# B&R Automation Studio project TD52 (part 49)

```iecst
	xMsg36[73].Enable	:=	IN_CU.tPB2MM.bParaSetupOk ;
	xMsg36[73].Set		:=	OUT_CU.bMsg3673;(* B3673 reserve operating message *)
	IF xMsg36[73].Set THEN iReset_Msg36[73] := iDelay_MsgAutoReset_100ms; ELSE iReset_Msg36[73] := LIMIT(0, iReset_Msg36[73] -1,32767); END_IF		(* activate 'Message Hold Time' to avoid log clathering by repeated OpMsg entries *)
	xMsg36[73].Reset 	:= 	(iReset_Msg36[73] < 1);		//.Reset := TRUE;
	xMsg36[73]();
	MM2VIS.bMsg3673		:=	xMsg36[73].Q;

	xMsg36[74].Enable	:=	IN_CU.tPB2MM.bParaSetupOk ;
	xMsg36[74].Set		:=	OUT_CU.bMsg3674;(* B3674 reserve operating message *)
	IF xMsg36[74].Set THEN iReset_Msg36[74] := iDelay_MsgAutoReset_100ms; ELSE iReset_Msg36[74] := LIMIT(0, iReset_Msg36[74] -1,32767); END_IF		(* activate 'Message Hold Time' to avoid log clathering by repeated OpMsg entries *)
	xMsg36[74].Reset 	:= 	(iReset_Msg36[74] < 1);		//.Reset := TRUE;
	xMsg36[74]();
	MM2VIS.bMsg3674		:=	xMsg36[74].Q;

	xMsg36[75].Enable	:=	IN_CU.tPB2MM.bParaSetupOk ;
	xMsg36[75].Set		:=	OUT_CU.bMsg3675;(* B3675 reserve operating message *)
	IF xMsg36[75].Set THEN iReset_Msg36[75] := iDelay_MsgAutoReset_100ms; ELSE iReset_Msg36[75] := LIMIT(0, iReset_Msg36[75] -1,32767); END_IF		(* activate 'Message Hold Time' to avoid log clathering by repeated OpMsg entries *)
	xMsg36[75].Reset 	:= 	(iReset_Msg36[75] < 1);		//.Reset := TRUE;
	xMsg36[75]();
	MM2VIS.bMsg3675		:=	xMsg36[75].Q;

	xMsg36[76].Enable	:=	IN_CU.tPB2MM.bParaSetupOk ;
	xMsg36[76].Set		:=	OUT_CU.bMsg3676;(* B3676 reserve operating message *)
	IF xMsg36[76].Set THEN iReset_Msg36[76] := iDelay_MsgAutoReset_100ms; ELSE iReset_Msg36[76] := LIMIT(0, iReset_Msg36[76] -1,32767); END_IF		(* activate 'Message Hold Time' to avoid log clathering by repeated OpMsg entries *)
	xMsg36[76].Reset 	:= 	(iReset_Msg36[76] < 1);		//.Reset := TRUE;
	xMsg36[76]();
	MM2VIS.bMsg3676		:=	xMsg36[76].Q;

	xMsg36[77].Enable	:=	IN_CU.tPB2MM.bParaSetupOk ;
	xMsg36[77].Set		:=	OUT_CU.bMsg3677;(* B3677 reserve operating message *)
	IF xMsg36[77].Set THEN iReset_Msg36[77] := iDelay_MsgAutoReset_100ms; ELSE iReset_Msg36[77] := LIMIT(0, iReset_Msg36[77] -1,32767); END_IF		(* activate 'Message Hold Time' to avoid log clathering by repeated OpMsg entries *)
	xMsg36[77].Reset 	:= 	(iReset_Msg36[77] < 1);		//.Reset := TRUE;
	xMsg36[77]();
	MM2VIS.bMsg3677		:=	xMsg36[77].Q;

	xMsg36[78].Enable	:=	IN_CU.tPB2MM.bParaSetupOk ;
	xMsg36[78].Set		:=	OUT_CU.bMsg3678;(* B3678 reserve operating message *)
	IF xMsg36[78].Set THEN iReset_Msg36[78] := iDelay_MsgAutoReset_100ms; ELSE iReset_Msg36[78] := LIMIT(0, iReset_Msg36[78] -1,32767); END_IF		(* activate 'Message Hold Time' to avoid log clathering by repeated OpMsg entries *)
	xMsg36[78].Reset 	:= 	(iReset_Msg36[78] < 1);		//.Reset := TRUE;
	xMsg36[78]();
	MM2VIS.bMsg3678		:=	xMsg36[78].Q;

	xMsg36[79].Enable	:=	IN_CU.tPB2MM.bParaSetupOk ;
	xMsg36[79].Set		:=	OUT_CU.bMsg3679;(* B3679 reserve operating message *)
	IF xMsg36[79].Set THEN iReset_Msg36[79] := iDelay_MsgAutoReset_100ms; ELSE iReset_Msg36[79] := LIMIT(0, iReset_Msg36[79] -1,32767); END_IF		(* activate 'Message Hold Time' to avoid log clathering by repeated OpMsg entries *)
	xMsg36[79].Reset 	:= 	(iReset_Msg36[79] < 1);		//.Reset := TRUE;
	xMsg36[79]();
	MM2VIS.bMsg3679		:=	xMsg36[79].Q;

	xMsg36[80].Enable	:=	IN_CU.tPB2MM.bParaSetupOk ;
	xMsg36[80].Set		:=	OUT_CU.bMsg3680;(* B3680 reserve operating message *)
	IF xMsg36[80].Set THEN iReset_Msg36[80] := iDelay_MsgAutoReset_100ms; ELSE iReset_Msg36[80] := LIMIT(0, iReset_Msg36[80] -1,32767); END_IF		(* activate 'Message Hold Time' to avoid log clathering by repeated OpMsg entries *)
	xMsg36[80].Reset 	:= 	(iReset_Msg36[80] < 1);		//.Reset := TRUE;
	xMsg36[80]();
	MM2VIS.bMsg3680		:=	xMsg36[80].Q;
	(*----------------------------------------------------------------------*)

	xMsg36[81].Enable	:=	IN_CU.tPB2MM.bParaSetupOk ;
	xMsg36[81].Set		:=	OUT_CU.bMsg3681;(* B3681 reserve operating message *)
	IF xMsg36[81].Set THEN iReset_Msg36[81] := iDelay_MsgAutoReset_100ms; ELSE iReset_Msg36[81] := LIMIT(0, iReset_Msg36[81] -1,32767); END_IF		(* activate 'Message Hold Time' to avoid log clathering by repeated OpMsg entries *)
	xMsg36[81].Reset 	:= 	(iReset_Msg36[81] < 1);		//.Reset := TRUE;
	xMsg36[81]();
	MM2VIS.bMsg3681		:=	xMsg36[81].Q;

	xMsg36[82].Enable	:=	IN_CU.tPB2MM.bParaSetupOk ;
	xMsg36[82].Set		:=	OUT_CU.bMsg3682;(* B3682 reserve operating message *)
	IF xMsg36[82].Set THEN iReset_Msg36[82] := iDelay_MsgAutoReset_100ms; ELSE iReset_Msg36[82] := LIMIT(0, iReset_Msg36[82] -1,32767); END_IF		(* activate 'Message Hold Time' to avoid log clathering by repeated OpMsg entries *)
	xMsg36[82].Reset 	:= 	(iReset_Msg36[82] < 1);		//.Reset := TRUE;
	xMsg36[82]();
	MM2VIS.bMsg3682		:=	xMsg36[82].Q;

	xMsg36[83].Enable	:=	IN_CU.tPB2MM.bParaSetupOk ;
	xMsg36[83].Set		:=	OUT_CU.bMsg3683;(* B3683 reserve operating message *)
	IF xMsg36[83].Set THEN iReset_Msg36[83] := iDelay_MsgAutoReset_100ms; ELSE iReset_Msg36[83] := LIMIT(0, iReset_Msg36[83] -1,32767); END_IF		(* activate 'Message Hold Time' to avoid log clathering by repeated OpMsg entries *)
	xMsg36[83].Reset 	:= 	(iReset_Msg36[83] < 1);		//.Reset := TRUE;
	xMsg36[83]();
	MM2VIS.bMsg3683		:=	xMsg36[83].Q;

	xMsg36[84].Enable	:=	IN_CU.tPB2MM.bParaSetupOk ;
	xMsg36[84].Set		:=	OUT_CU.bMsg3684;(* B3684 reserve operating message *)
	IF xMsg36[84].Set THEN iReset_Msg36[84] := iDelay_MsgAutoReset_100ms; ELSE iReset_Msg36[84] := LIMIT(0, iReset_Msg36[84] -1,32767); END_IF		(* activate 'Message Hold Time' to avoid log clathering by repeated OpMsg entries *)
	xMsg36[84].Reset 	:= 	(iReset_Msg36[84] < 1);		//.Reset := TRUE;
	xMsg36[84]();
	MM2VIS.bMsg3684		:=	xMsg36[84].Q;

	xMsg36[85].Enable	:=	IN_CU.tPB2MM.bParaSetupOk ;
	xMsg36[85].Set		:=	OUT_CU.bMsg3685;(* B3685 reserve operating message *)
	IF xMsg36[85].Set THEN iReset_Msg36[85] := iDelay_MsgAutoReset_100ms; ELSE iReset_Msg36[85] := LIMIT(0, iReset_Msg36[85] -1,32767); END_IF		(* activate 'Message Hold Time' to avoid log clathering by repeated OpMsg entries *)
	xMsg36[85].Reset 	:= 	(iReset_Msg36[85] < 1);		//.Reset := TRUE;
	xMsg36[85]();
	MM2VIS.bMsg3685		:=	xMsg36[85].Q;

	xMsg36[86].Enable	:=	IN_CU.tPB2MM.bParaSetupOk ;
	xMsg36[86].Set		:=	OUT_CU.bMsg3686;(* B3686 reserve operating message *)
	IF xMsg36[86].Set THEN iReset_Msg36[86] := iDelay_MsgAutoReset_100ms; ELSE iReset_Msg36[86] := LIMIT(0, iReset_Msg36[86] -1,32767); END_IF		(* activate 'Message Hold Time' to avoid log clathering by repeated OpMsg entries *)
	xMsg36[86].Reset 	:= 	(iReset_Msg36[86] < 1);		//.Reset := TRUE;
	xMsg36[86]();
	MM2VIS.bMsg3686		:=	xMsg36[86].Q;

	xMsg36[87].Enable	:=	IN_CU.tPB2MM.bParaSetupOk ;
	xMsg36[87].Set		:=	OUT_CU.bMsg3687;(* B3687 reserve operating message *)
	IF xMsg36[87].Set THEN iReset_Msg36[87] := iDelay_MsgAutoReset_100ms; ELSE iReset_Msg36[87] := LIMIT(0, iReset_Msg36[87] -1,32767); END_IF		(* activate 'Message Hold Time' to avoid log clathering by repeated OpMsg entries *)
	xMsg36[87].Reset 	:= 	(iReset_Msg36[87] < 1);		//.Reset := TRUE;
	xMsg36[87]();
	MM2VIS.bMsg3687		:=	xMsg36[87].Q;

	xMsg36[88].Enable	:=	IN_CU.tPB2MM.bParaSetupOk ;
	xMsg36[88].Set		:=	OUT_CU.bMsg3688;(* B3688 reserve operating message *)
	IF xMsg36[88].Set THEN iReset_Msg36[88] := iDelay_MsgAutoReset_100ms; ELSE iReset_Msg36[88] := LIMIT(0, iReset_Msg36[88] -1,32767); END_IF		(* activate 'Message Hold Time' to avoid log clathering by repeated OpMsg entries *)
	xMsg36[88].Reset 	:= 	(iReset_Msg36[88] < 1);		//.Reset := TRUE;
	xMsg36[88]();
	MM2VIS.bMsg3688		:=	xMsg36[88].Q;

	xMsg36[89].Enable	:=	IN_CU.tPB2MM.bParaSetupOk ;
	xMsg36[89].Set		:=	OUT_CU.bMsg3689;(* B3689 reserve operating message *)
	IF xMsg36[89].Set THEN iReset_Msg36[89] := iDelay_MsgAutoReset_100ms; ELSE iReset_Msg36[89] := LIMIT(0, iReset_Msg36[89] -1,32767); END_IF		(* activate 'Message Hold Time' to avoid log clathering by repeated OpMsg entries *)
	xMsg36[89].Reset 	:= 	(iReset_Msg36[89] < 1);		//.Reset := TRUE;
	xMsg36[89]();
	MM2VIS.bMsg3689		:=	xMsg36[89].Q;

	xMsg36[90].Enable	:=	IN_CU.tPB2MM.bParaSetupOk ;
	xMsg36[90].Set		:=	OUT_CU.bMsg3690;(* B3690 reserve operating message *)
	IF xMsg36[90].Set THEN iReset_Msg36[90] := iDelay_MsgAutoReset_100ms; ELSE iReset_Msg36[90] := LIMIT(0, iReset_Msg36[90] -1,32767); END_IF		(* activate 'Message Hold Time' to avoid log clathering by repeated OpMsg entries *)
	xMsg36[90].Reset 	:= 	(iReset_Msg36[90] < 1);		//.Reset := TRUE;
	xMsg36[90]();
	MM2VIS.bMsg3690		:=	xMsg36[90].Q;
	(*----------------------------------------------------------------------*)

	xMsg36[91].Enable	:=	IN_CU.tPB2MM.bParaSetupOk ;
	xMsg36[91].Set		:=	OUT_CU.bMsg3691;(* B3691 reserve operating message *)
	IF xMsg36[91].Set THEN iReset_Msg36[91] := iDelay_MsgAutoReset_100ms; ELSE iReset_Msg36[91] := LIMIT(0, iReset_Msg36[91] -1,32767); END_IF		(* activate 'Message Hold Time' to avoid log clathering by repeated OpMsg entries *)
	xMsg36[91].Reset 	:= 	(iReset_Msg36[91] < 1);		//.Reset := TRUE;
	xMsg36[91]();
	MM2VIS.bMsg3691		:=	xMsg36[91].Q;

	xMsg36[92].Enable	:=	IN_CU.tPB2MM.bParaSetupOk ;
	xMsg36[92].Set		:=	OUT_CU.bMsg3692;(* B3692 reserve operating message *)
	IF xMsg36[92].Set THEN iReset_Msg36[92] := iDelay_MsgAutoReset_100ms; ELSE iReset_Msg36[92] := LIMIT(0, iReset_Msg36[92] -1,32767); END_IF		(* activate 'Message Hold Time' to avoid log clathering by repeated OpMsg entries *)
	xMsg36[92].Reset 	:= 	(iReset_Msg36[92] < 1);		//.Reset := TRUE;
	xMsg36[92]();
	MM2VIS.bMsg3692		:=	xMsg36[92].Q;

	xMsg36[93].Enable	:=	IN_CU.tPB2MM.bParaSetupOk ;
	xMsg36[93].Set		:=	OUT_CU.bMsg3693;(* B3693 reserve operating message *)
	IF xMsg36[93].Set THEN iReset_Msg36[93] := iDelay_MsgAutoReset_100ms; ELSE iReset_Msg36[93] := LIMIT(0, iReset_Msg36[93] -1,32767); END_IF		(* activate 'Message Hold Time' to avoid log clathering by repeated OpMsg entries *)
	xMsg36[93].Reset 	:= 	(iReset_Msg36[93] < 1);		//.Reset := TRUE;
	xMsg36[93]();
	MM2VIS.bMsg3693		:=	xMsg36[93].Q;

	xMsg36[94].Enable	:=	IN_CU.tPB2MM.bParaSetupOk ;
	xMsg36[94].Set		:=	OUT_CU.bMsg3694;(* B3694 reserve operating message *)
	IF xMsg36[94].Set THEN iReset_Msg36[94] := iDelay_MsgAutoReset_100ms; ELSE iReset_Msg36[94] := LIMIT(0, iReset_Msg36[94] -1,32767); END_IF		(* activate 'Message Hold Time' to avoid log clathering by repeated OpMsg entries *)
	xMsg36[94].Reset 	:= 	(iReset_Msg36[94] < 1);		//.Reset := TRUE;
	xMsg36[94]();
	MM2VIS.bMsg3694		:=	xMsg36[94].Q;

	xMsg36[95].Enable	:=	IN_CU.tPB2MM.bParaSetupOk ;
	xMsg36[95].Set		:=	OUT_CU.bMsg3695;(* B3695 reserve operating message *)
	IF xMsg36[95].Set THEN iReset_Msg36[95] := iDelay_MsgAutoReset_100ms; ELSE iReset_Msg36[95] := LIMIT(0, iReset_Msg36[95] -1,32767); END_IF		(* activate 'Message Hold Time' to avoid log clathering by repeated OpMsg entries *)
	xMsg36[95].Reset 	:= 	(iReset_Msg36[95] < 1);		//.Reset := TRUE;
	xMsg36[95]();
	MM2VIS.bMsg3695		:=	xMsg36[95].Q;

	xMsg36[96].Enable	:=	IN_CU.tPB2MM.bParaSetupOk ;
	xMsg36[96].Set		:=	OUT_CU.bMsg3696;(* B3696 reserve operating message *)
	IF xMsg36[96].Set THEN iReset_Msg36[96] := iDelay_MsgAutoReset_100ms; ELSE iReset_Msg36[96] := LIMIT(0, iReset_Msg36[96] -1,32767); END_IF		(* activate 'Message Hold Time' to avoid log clathering by repeated OpMsg entries *)
	xMsg36[96].Reset 	:= 	(iReset_Msg36[96] < 1);		//.Reset := TRUE;
	xMsg36[96]();
	MM2VIS.bMsg3696		:=	xMsg36[96].Q;

	xMsg36[97].Enable	:=	IN_CU.tPB2MM.bParaSetupOk ;
	xMsg36[97].Set		:=	OUT_CU.bMsg3697;(* B3697 reserve operating message *)
	IF xMsg36[97].Set THEN iReset_Msg36[97] := iDelay_MsgAutoReset_100ms; ELSE iReset_Msg36[97] := LIMIT(0, iReset_Msg36[97] -1,32767); END_IF		(* activate 'Message Hold Time' to avoid log clathering by repeated OpMsg entries *)
	xMsg36[97].Reset 	:= 	(iReset_Msg36[97] < 1);		//.Reset := TRUE;
	xMsg36[97]();
	MM2VIS.bMsg3697		:=	xMsg36[97].Q;

	xMsg36[98].Enable	:=	IN_CU.tPB2MM.bParaSetupOk ;
	xMsg36[98].Set		:=	OUT_CU.bMsg3698;(* B3698 reserve operating message *)
	IF xMsg36[98].Set THEN iReset_Msg36[98] := iDelay_MsgAutoReset_100ms; ELSE iReset_Msg36[98] := LIMIT(0, iReset_Msg36[98] -1,32767); END_IF		(* activate 'Message Hold Time' to avoid log clathering by repeated OpMsg entries *)
	xMsg36[98].Reset 	:= 	(iReset_Msg36[98] < 1);		//.Reset := TRUE;
	xMsg36[98]();
	MM2VIS.bMsg3698		:=	xMsg36[98].Q;

	xMsg36[99].Enable	:=	IN_CU.tPB2MM.bParaSetupOk ;
	xMsg36[99].Set		:=	OUT_CU.bMsg3699;(* B3699 reserve operating message *)
	IF xMsg36[99].Set THEN iReset_Msg36[99] := iDelay_MsgAutoReset_100ms; ELSE iReset_Msg36[99] := LIMIT(0, iReset_Msg36[99] -1,32767); END_IF		(* activate 'Message Hold Time' to avoid log clathering by repeated OpMsg entries *)
	xMsg36[99].Reset 	:= 	(iReset_Msg36[99] < 1);		//.Reset := TRUE;
	xMsg36[99]();
	MM2VIS.bMsg3699		:=	xMsg36[99].Q;

	xMsg3700.Enable		:=	IN_CU.tPB2MM.bParaSetupOk ;
	xMsg3700.Set		:=	OUT_CU.bMsg3700;(* B3700 reserve operating message *)
	IF xMsg3700.Set THEN iReset_Msg3700 := iDelay_MsgAutoReset_100ms; ELSE iReset_Msg3700 := LIMIT(0, iReset_Msg3700 -1,32767); END_IF		(* activate 'Message Hold Time' to avoid log clathering by repeated OpMsg entries *)
	xMsg3700.Reset 	:= 	(iReset_Msg3700 < 1);		//.Reset := TRUE;
	xMsg3700();
	MM2VIS.bMsg3700		:=	xMsg3700.Q;

	(* W6701 to W6799:  reserve operating message 109 - 207 *) (*import HMI Extension *)
	FOR cnt := 01 TO 99 DO
		(*set standard message options*)
		xMsg67[cnt].Enable	:= 	IN_CU.tPB2MM.bParaSetupOk ;
		IF xMsg67[cnt].Set THEN iReset_Msg67[cnt] := iDelay_MsgAutoReset_100ms; ELSE iReset_Msg67[cnt] := LIMIT(0, iReset_Msg67[cnt] -1,32767); END_IF		(* activate 'Message Hold Time' to avoid log clathering by repeated OpMsg entries *)
		xMsg67[cnt].Reset 	:= 	(iReset_Msg67[cnt] < 1);		//.Reset := TRUE;
		xMsg67[cnt]();	(*function call*)
	END_FOR

	xMsg67[01].Set		:=	OUT_CU.bMsg6701;(* B6701 reserve operating message 109 *) (*import HMI Extension *)
	MM2VIS.bMsg6701		:=	xMsg67[01].Q;

	xMsg67[02].Set		:=	OUT_CU.bMsg6702;(* B6702 reserve operating message 110 *) (*import HMI Extension *)
	MM2VIS.bMsg6702		:=	xMsg67[02].Q;

	xMsg67[03].Set		:=	OUT_CU.bMsg6703;(* B6703 reserve operating message 111 *) (*import HMI Extension *)
	MM2VIS.bMsg6703		:=	xMsg67[03].Q;

	xMsg67[04].Set		:=	OUT_CU.bMsg6704;(* B6704 reserve operating message 112 *) (*import HMI Extension *)
	MM2VIS.bMsg6704		:=	xMsg67[04].Q;

	xMsg67[05].Set		:=	OUT_CU.bMsg6705;(* B6705 reserve operating message 113 *) (*import HMI Extension *)
	MM2VIS.bMsg6705		:=	xMsg67[05].Q;

	xMsg67[06].Set		:=	OUT_CU.bMsg6706;(* B6706 reserve operating message 114 *) (*import HMI Extension *)
	MM2VIS.bMsg6706		:=	xMsg67[06].Q;

	xMsg67[07].Set		:=	OUT_CU.bMsg6707;(* B6707 reserve operating message 115 *) (*import HMI Extension *)
	MM2VIS.bMsg6707		:=	xMsg67[07].Q;

	xMsg67[08].Set		:=	OUT_CU.bMsg6708;(* B6708 reserve operating message 116 *) (*import HMI Extension *)
	MM2VIS.bMsg6708		:=	xMsg67[08].Q;

	xMsg67[09].Set		:=	OUT_CU.bMsg6709;(* B6709 reserve operating message 117 *) (*import HMI Extension *)
	MM2VIS.bMsg6709		:=	xMsg67[09].Q;

	xMsg67[10].Set		:=	OUT_CU.bMsg6710;(* B6710 reserve operating message 118 *) (*import HMI Extension *)
	MM2VIS.bMsg6710		:=	xMsg67[10].Q;

	xMsg67[11].Set		:=	OUT_CU.bMsg6711;(* B6711 reserve operating message 119 *) (*import HMI Extension *)
	MM2VIS.bMsg6711		:=	xMsg67[11].Q;

	xMsg67[12].Set		:=	OUT_CU.bMsg6712;(* B6712 reserve operating message 120 *) (*import HMI Extension *)
	MM2VIS.bMsg6712		:=	xMsg67[12].Q;

	xMsg67[13].Set		:=	OUT_CU.bMsg6713;(* B6713 reserve operating message 121 *) (*import HMI Extension *)
	MM2VIS.bMsg6713		:=	xMsg67[13].Q;

	xMsg67[14].Set		:=	OUT_CU.bMsg6714;(* B6714 reserve operating message 122 *) (*import HMI Extension *)
	MM2VIS.bMsg6714		:=	xMsg67[14].Q;

	xMsg67[15].Set		:=	OUT_CU.bMsg6715;(* B6715 reserve operating message 123 *) (*import HMI Extension *)
	MM2VIS.bMsg6715		:=	xMsg67[15].Q;

	xMsg67[16].Set		:=	OUT_CU.bMsg6716;(* B6716 reserve operating message 124 *) (*import HMI Extension *)
	MM2VIS.bMsg6716		:=	xMsg67[16].Q;

	xMsg67[17].Set		:=	OUT_CU.bMsg6717;(* B6717 reserve operating message 125 *) (*import HMI Extension *)
	MM2VIS.bMsg6717		:=	xMsg67[17].Q;

	xMsg67[18].Set		:=	OUT_CU.bMsg6718;(* B6718 reserve operating message 126 *) (*import HMI Extension *)
	MM2VIS.bMsg6718		:=	xMsg67[18].Q;

	xMsg67[19].Set		:=	OUT_CU.bMsg6719;(* B6719 reserve operating message 127 *) (*import HMI Extension *)
	MM2VIS.bMsg6719		:=	xMsg67[19].Q;

	xMsg67[20].Set		:=	OUT_CU.bMsg6720;(* B6720 reserve operating message 128 *) (*import HMI Extension *)
	MM2VIS.bMsg6720		:=	xMsg67[20].Q;

	xMsg67[21].Set		:=	OUT_CU.bMsg6721;(* B6721 reserve operating message 129 *) (*import HMI Extension *)
	MM2VIS.bMsg6721		:=	xMsg67[21].Q;

	xMsg67[22].Set		:=	OUT_CU.bMsg6722;(* B6722 reserve operating message 130 *) (*import HMI Extension *)
	MM2VIS.bMsg6722		:=	xMsg67[22].Q;

	xMsg67[23].Set		:=	OUT_CU.bMsg6723;(* B6723 reserve operating message 131 *) (*import HMI Extension *)
	MM2VIS.bMsg6723		:=	xMsg67[23].Q;

	xMsg67[24].Set		:=	OUT_CU.bMsg6724;(* B6724 reserve operating message 132 *) (*import HMI Extension *)
	MM2VIS.bMsg6724		:=	xMsg67[24].Q;

	xMsg67[25].Set		:=	OUT_CU.bMsg6725;(* B6725 reserve operating message 133 *) (*import HMI Extension *)
	MM2VIS.bMsg6725		:=	xMsg67[25].Q;

	xMsg67[26].Set		:=	OUT_CU.bMsg6726;(* B6726 reserve operating message 134 *) (*import HMI Extension *)
	MM2VIS.bMsg6726		:=	xMsg67[26].Q;

	xMsg67[27].Set		:=	OUT_CU.bMsg6727;(* B6727 reserve operating message 135 *) (*import HMI Extension *)
	MM2VIS.bMsg6727		:=	xMsg67[27].Q;

	xMsg67[28].Set		:=	OUT_CU.bMsg6728;(* B6728 reserve operating message 136 *) (*import HMI Extension *)
	MM2VIS.bMsg6728		:=	xMsg67[28].Q;

	xMsg67[29].Set		:=	OUT_CU.bMsg6729;(* B6729 reserve operating message 137 *) (*import HMI Extension *)
	MM2VIS.bMsg6729		:=	xMsg67[29].Q;

	xMsg67[30].Set		:=	OUT_CU.bMsg6730;(* B6730 reserve operating message 138 *) (*import HMI Extension *)
	MM2VIS.bMsg6730		:=	xMsg67[30].Q;

	xMsg67[31].Set		:=	OUT_CU.bMsg6731;(* B6731 reserve operating message 139 *) (*import HMI Extension *)
	MM2VIS.bMsg6731		:=	xMsg67[31].Q;

	xMsg67[32].Set		:=	OUT_CU.bMsg6732;(* B6732 reserve operating message 140 *) (*import HMI Extension *)
	MM2VIS.bMsg6732		:=	xMsg67[32].Q;

	xMsg67[33].Set		:=	OUT_CU.bMsg6733;(* B6733 reserve operating message 141 *) (*import HMI Extension *)
	MM2VIS.bMsg6733		:=	xMsg67[33].Q;

	xMsg67[34].Set		:=	OUT_CU.bMsg6734;(* B6734 reserve operating message 142 *) (*import HMI Extension *)
	MM2VIS.bMsg6734		:=	xMsg67[34].Q;

	xMsg67[35].Set		:=	OUT_CU.bMsg6735;(* B6735 reserve operating message 143 *) (*import HMI Extension *)
	MM2VIS.bMsg6735		:=	xMsg67[35].Q;

	xMsg67[36].Set		:=	OUT_CU.bMsg6736;(* B6736 reserve operating message 144 *) (*import HMI Extension *)
	MM2VIS.bMsg6736		:=	xMsg67[36].Q;

	xMsg67[37].Set		:=	OUT_CU.bMsg6737;(* B6737 reserve operating message 145 *) (*import HMI Extension *)
	MM2VIS.bMsg6737		:=	xMsg67[37].Q;

	xMsg67[38].Set		:=	OUT_CU.bMsg6738;(* B6738 reserve operating message 146 *) (*import HMI Extension *)
	MM2VIS.bMsg6738		:=	xMsg67[38].Q;

	xMsg67[39].Set		:=	OUT_CU.bMsg6739;(* B6739 reserve operating message 147 *) (*import HMI Extension *)
	MM2VIS.bMsg6739		:=	xMsg67[39].Q;

	xMsg67[40].Set		:=	OUT_CU.bMsg6740;(* B6740 reserve operating message 148 *) (*import HMI Extension *)
	MM2VIS.bMsg6740		:=	xMsg67[40].Q;

	xMsg67[41].Set		:=	OUT_CU.bMsg6741;(* B6741 reserve operating message 149 *) (*import HMI Extension *)
	MM2VIS.bMsg6741		:=	xMsg67[41].Q;

	xMsg67[42].Set		:=	OUT_CU.bMsg6742;(* B6742 reserve operating message 150 *) (*import HMI Extension *)
	MM2VIS.bMsg6742		:=	xMsg67[42].Q;

	xMsg67[43].Set		:=	OUT_CU.bMsg6743;(* B6743 reserve operating message 151 *) (*import HMI Extension *)
	MM2VIS.bMsg6743		:=	xMsg67[43].Q;

	xMsg67[44].Set		:=	OUT_CU.bMsg6744;(* B6744 reserve operating message 152 *) (*import HMI Extension *)
	MM2VIS.bMsg6744		:=	xMsg67[44].Q;

	xMsg67[45].Set		:=	OUT_CU.bMsg6745;(* B6745 reserve operating message 153 *) (*import HMI Extension *)
	MM2VIS.bMsg6745		:=	xMsg67[45].Q;

	xMsg67[46].Set		:=	OUT_CU.bMsg6746;(* B6746 reserve operating message 154 *) (*import HMI Extension *)
	MM2VIS.bMsg6746		:=	xMsg67[46].Q;

	xMsg67[47].Set		:=	OUT_CU.bMsg6747;(* B6747 reserve operating message 155 *) (*import HMI Extension *)
	MM2VIS.bMsg6747		:=	xMsg67[47].Q;

	xMsg67[48].Set		:=	OUT_CU.bMsg6748;(* B6748 reserve operating message 156 *) (*import HMI Extension *)
	MM2VIS.bMsg6748		:=	xMsg67[48].Q;

	xMsg67[49].Set		:=	OUT_CU.bMsg6749;(* B6749 reserve operating message 157 *) (*import HMI Extension *)
	MM2VIS.bMsg6749		:=	xMsg67[49].Q;

	xMsg67[50].Set		:=	OUT_CU.bMsg6750;(* B6750 reserve operating message 158 *) (*import HMI Extension *)
	MM2VIS.bMsg6750		:=	xMsg67[50].Q;

	xMsg67[51].Set		:=	OUT_CU.bMsg6751;(* B6751 reserve operating message 159 *) (*import HMI Extension *)
	MM2VIS.bMsg6751		:=	xMsg67[51].Q;

	xMsg67[52].Set		:=	OUT_CU.bMsg6752;(* B6752 reserve operating message 160 *) (*import HMI Extension *)
	MM2VIS.bMsg6752		:=	xMsg67[52].Q;

	xMsg67[53].Set		:=	OUT_CU.bMsg6753;(* B6753 reserve operating message 161 *) (*import HMI Extension *)
	MM2VIS.bMsg6753		:=	xMsg67[53].Q;

	xMsg67[54].Set		:=	OUT_CU.bMsg6754;(* B6754 reserve operating message 162 *) (*import HMI Extension *)
	MM2VIS.bMsg6754		:=	xMsg67[54].Q;

	xMsg67[55].Set		:=	OUT_CU.bMsg6755;(* B6755 reserve operating message 163 *) (*import HMI Extension *)
	MM2VIS.bMsg6755		:=	xMsg67[55].Q;

	xMsg67[56].Set		:=	OUT_CU.bMsg6756;(* B6756 reserve operating message 164 *) (*import HMI Extension *)
	MM2VIS.bMsg6756		:=	xMsg67[56].Q;

	xMsg67[57].Set		:=	OUT_CU.bMsg6757;(* B6757 reserve operating message 165 *) (*import HMI Extension *)
	MM2VIS.bMsg6757		:=	xMsg67[57].Q;

	xMsg67[58].Set		:=	OUT_CU.bMsg6758;(* B6758 reserve operating message 166 *) (*import HMI Extension *)
	MM2VIS.bMsg6758		:=	xMsg67[58].Q;

	xMsg67[59].Set		:=	OUT_CU.bMsg6759;(* B6759 reserve operating message 167 *) (*import HMI Extension *)
	MM2VIS.bMsg6759		:=	xMsg67[59].Q;

	xMsg67[60].Set		:=	OUT_CU.bMsg6760;(* B6760 reserve operating message 168 *) (*import HMI Extension *)
	MM2VIS.bMsg6760		:=	xMsg67[60].Q;

	xMsg67[61].Set		:=	OUT_CU.bMsg6761;(* B6761 reserve operating message 169 *) (*import HMI Extension *)
	MM2VIS.bMsg6761		:=	xMsg67[61].Q;

	xMsg67[62].Set		:=	OUT_CU.bMsg6762;(* B6762 reserve operating message 170 *) (*import HMI Extension *)
	MM2VIS.bMsg6762		:=	xMsg67[62].Q;

	xMsg67[63].Set		:=	OUT_CU.bMsg6763;(* B6763 reserve operating message 171 *) (*import HMI Extension *)
	MM2VIS.bMsg6763		:=	xMsg67[63].Q;

	xMsg67[64].Set		:=	OUT_CU.bMsg6764;(* B6764 reserve operating message 172 *) (*import HMI Extension *)
	MM2VIS.bMsg6764		:=	xMsg67[64].Q;

	xMsg67[65].Set		:=	OUT_CU.bMsg6765;(* B6765 reserve operating message 173 *) (*import HMI Extension *)
	MM2VIS.bMsg6765		:=	xMsg67[65].Q;

	xMsg67[66].Set		:=	OUT_CU.bMsg6766;(* B6766 reserve operating message 174 *) (*import HMI Extension *)
	MM2VIS.bMsg6766		:=	xMsg67[66].Q;

	xMsg67[67].Set		:=	OUT_CU.bMsg6767;(* B6767 reserve operating message 175 *) (*import HMI Extension *)
	MM2VIS.bMsg6767		:=	xMsg67[67].Q;

	xMsg67[68].Set		:=	OUT_CU.bMsg6768;(* B6768 reserve operating message 176 *) (*import HMI Extension *)
	MM2VIS.bMsg6768		:=	xMsg67[68].Q;

	xMsg67[69].Set		:=	OUT_CU.bMsg6769;(* B6769 reserve operating message 177 *) (*import HMI Extension *)
	MM2VIS.bMsg6769		:=	xMsg67[69].Q;

	xMsg67[70].Set		:=	OUT_CU.bMsg6770;(* B6770 reserve operating message 178 *) (*import HMI Extension *)
	MM2VIS.bMsg6770		:=	xMsg67[70].Q;

	xMsg67[71].Set		:=	OUT_CU.bMsg6771;(* B6771 reserve operating message 179 *) (*import HMI Extension *)
	MM2VIS.bMsg6771		:=	xMsg67[71].Q;

	xMsg67[72].Set		:=	OUT_CU.bMsg6772;(* B6772 reserve operating message 180 *) (*import HMI Extension *)
	MM2VIS.bMsg6772		:=	xMsg67[72].Q;

	xMsg67[73].Set		:=	OUT_CU.bMsg6773;(* B6773 reserve operating message 181 *) (*import HMI Extension *)
	MM2VIS.bMsg6773		:=	xMsg67[73].Q;

	xMsg67[74].Set		:=	OUT_CU.bMsg6774;(* B6774 reserve operating message 182 *) (*import HMI Extension *)
	MM2VIS.bMsg6774		:=	xMsg67[74].Q;

	xMsg67[75].Set		:=	OUT_CU.bMsg6775;(* B6775 reserve operating message 183 *) (*import HMI Extension *)
	MM2VIS.bMsg6775		:=	xMsg67[75].Q;

	xMsg67[76].Set		:=	OUT_CU.bMsg6776;(* B6776 reserve operating message 184 *) (*import HMI Extension *)
	MM2VIS.bMsg6776		:=	xMsg67[76].Q;

	xMsg67[77].Set		:=	OUT_CU.bMsg6777;(* B6777 reserve operating message 185 *) (*import HMI Extension *)
	MM2VIS.bMsg6777		:=	xMsg67[77].Q;

	xMsg67[78].Set		:=	OUT_CU.bMsg6778;(* B6778 reserve operating message 186 *) (*import HMI Extension *)
	MM2VIS.bMsg6778		:=	xMsg67[78].Q;

	xMsg67[79].Set		:=	OUT_CU.bMsg6779;(* B6779 reserve operating message 187 *) (*import HMI Extension *)
	MM2VIS.bMsg6779		:=	xMsg67[79].Q;

	xMsg67[80].Set		:=	OUT_CU.bMsg6780;(* B6780 reserve operating message 188 *) (*import HMI Extension *)
	MM2VIS.bMsg6780		:=	xMsg67[80].Q;

	xMsg67[81].Set		:=	OUT_CU.bMsg6781;(* B6781 reserve operating message 189 *) (*import HMI Extension *)
	MM2VIS.bMsg6781		:=	xMsg67[81].Q;

	xMsg67[82].Set		:=	OUT_CU.bMsg6782;(* B6782 reserve operating message 190 *) (*import HMI Extension *)
	MM2VIS.bMsg6782		:=	xMsg67[82].Q;

	xMsg67[83].Set		:=	OUT_CU.bMsg6783;(* B6783 reserve operating message 191 *) (*import HMI Extension *)
	MM2VIS.bMsg6783		:=	xMsg67[83].Q;

	xMsg67[84].Set		:=	OUT_CU.bMsg6784;(* B6784 reserve operating message 192 *) (*import HMI Extension *)
	MM2VIS.bMsg6784		:=	xMsg67[84].Q;

	xMsg67[85].Set		:=	OUT_CU.bMsg6785;(* B6785 reserve operating message 193 *) (*import HMI Extension *)
	MM2VIS.bMsg6785		:=	xMsg67[85].Q;

	xMsg67[86].Set		:=	OUT_CU.bMsg6786;(* B6786 reserve operating message 194 *) (*import HMI Extension *)
	MM2VIS.bMsg6786		:=	xMsg67[86].Q;

	xMsg67[87].Set		:=	OUT_CU.bMsg6787;(* B6787 reserve operating message 195 *) (*import HMI Extension *)
	MM2VIS.bMsg6787		:=	xMsg67[87].Q;

	xMsg67[88].Set		:=	OUT_CU.bMsg6788;(* B6788 reserve operating message 196 *) (*import HMI Extension *)
	MM2VIS.bMsg6788		:=	xMsg67[88].Q;

	xMsg67[89].Set		:=	OUT_CU.bMsg6789;(* B6789 reserve operating message 197 *) (*import HMI Extension *)
	MM2VIS.bMsg6789		:=	xMsg67[89].Q;

	xMsg67[90].Set		:=	OUT_CU.bMsg6790;(* B6790 reserve operating message 198 *) (*import HMI Extension *)
	MM2VIS.bMsg6790		:=	xMsg67[90].Q;

	xMsg67[91].Set		:=	OUT_CU.bMsg6791;(* B6791 reserve operating message 199 *) (*import HMI Extension *)
	MM2VIS.bMsg6791		:=	xMsg67[91].Q;

	xMsg67[92].Set		:=	OUT_CU.bMsg6792;(* B6792 reserve operating message 200 *) (*import HMI Extension *)
	MM2VIS.bMsg6792		:=	xMsg67[92].Q;

	xMsg67[93].Set		:=	OUT_CU.bMsg6793;(* B6793 reserve operating message 201 *) (*import HMI Extension *)
	MM2VIS.bMsg6793		:=	xMsg67[93].Q;

	xMsg67[94].Set		:=	OUT_CU.bMsg6794;(* B6794 reserve operating message 202 *) (*import HMI Extension *)
	MM2VIS.bMsg6794		:=	xMsg67[94].Q;

	xMsg67[95].Set		:=	OUT_CU.bMsg6795;(* B6795 reserve operating message 203 *) (*import HMI Extension *)
	MM2VIS.bMsg6795		:=	xMsg67[95].Q;

	xMsg67[96].Set		:=	OUT_CU.bMsg6796;(* B6796 reserve operating message 204 *) (*import HMI Extension *)
	MM2VIS.bMsg6796		:=	xMsg67[96].Q;

	xMsg67[97].Set		:=	OUT_CU.bMsg6797;(* B6797 reserve operating message 205 *) (*import HMI Extension *)
	MM2VIS.bMsg6797		:=	xMsg67[97].Q;

	xMsg67[98].Set		:=	OUT_CU.bMsg6798;(* B6798 reserve operating message 206 *) (*import HMI Extension *)
	MM2VIS.bMsg6798		:=	xMsg67[98].Q;

	xMsg67[99].Set		:=	OUT_CU.bMsg6799;(* B6799 reserve operating message 207 *) (*import HMI Extension *)
	MM2VIS.bMsg6799		:=	xMsg67[99].Q;

//	xMsg67[100].Set		//	MOVED TO xMsg68[0].Set
//	MM2VIS.bMsg6800		//	MOVED TO xMsg68[0].Set

	(* W6800 to W6899:  reserve operating message 208 - 307 *) (*import HMI Extension *)
	FOR cnt := 00 TO 99 DO
		(*set standard message options*)
		xMsg68[cnt].Enable	:= 	IN_CU.tPB2MM.bParaSetupOk ;
		IF xMsg68[cnt].Set THEN iReset_Msg68[cnt] := iDelay_MsgAutoReset_100ms; ELSE iReset_Msg68[cnt] := LIMIT(0, iReset_Msg68[cnt] -1,32767); END_IF		(* activate 'Message Hold Time' to avoid log clathering by repeated OpMsg entries *)
		xMsg68[cnt].Reset 	:= 	(iReset_Msg68[cnt] < 1);		//.Reset := TRUE;
		xMsg68[cnt]();	(*function call*)
	END_FOR

	xMsg68[0].Set		:=	OUT_CU.bMsg6800;(* B6800 reserve operating message 208 *) (*import HMI Extension *)
	MM2VIS.bMsg6800		:=	xMsg68[0].Q;

	xMsg68[01].Set		:=	OUT_CU.bMsg6801;(* B6801 reserve operating message 209 *) (*import HMI Extension *)
	MM2VIS.bMsg6801		:=	xMsg68[01].Q;

	xMsg68[02].Set		:=	OUT_CU.bMsg6802;(* B6802 reserve operating message 210 *) (*import HMI Extension *)
	MM2VIS.bMsg6802		:=	xMsg68[02].Q;

	xMsg68[03].Set		:=	OUT_CU.bMsg6803;(* B6803 reserve operating message 211 *) (*import HMI Extension *)
	MM2VIS.bMsg6803		:=	xMsg68[03].Q;

	xMsg68[04].Set		:=	OUT_CU.bMsg6804;(* B6804 reserve operating message 212 *) (*import HMI Extension *)
	MM2VIS.bMsg6804		:=	xMsg68[04].Q;

	xMsg68[05].Set		:=	OUT_CU.bMsg6805;(* B6805 reserve operating message 213 *) (*import HMI Extension *)
	MM2VIS.bMsg6805		:=	xMsg68[05].Q;

	xMsg68[06].Set		:=	OUT_CU.bMsg6806;(* B6806 reserve operating message 214 *) (*import HMI Extension *)
	MM2VIS.bMsg6806		:=	xMsg68[06].Q;

	xMsg68[07].Set		:=	OUT_CU.bMsg6807;(* B6807 reserve operating message 215 *) (*import HMI Extension *)
	MM2VIS.bMsg6807		:=	xMsg68[07].Q;

	xMsg68[08].Set		:=	OUT_CU.bMsg6808;(* B6808 reserve operating message 216 *) (*import HMI Extension *)
	MM2VIS.bMsg6808		:=	xMsg68[08].Q;

	xMsg68[09].Set		:=	OUT_CU.bMsg6809;(* B6809 reserve operating message 217 *) (*import HMI Extension *)
	MM2VIS.bMsg6809		:=	xMsg68[09].Q;

	xMsg68[10].Set		:=	OUT_CU.bMsg6810;(* B6810 reserve operating message 218 *) (*import HMI Extension *)
	MM2VIS.bMsg6810		:=	xMsg68[10].Q;

	xMsg68[11].Set		:=	OUT_CU.bMsg6811;(* B6811 reserve operating message 219 *) (*import HMI Extension *)
	MM2VIS.bMsg6811		:=	xMsg68[11].Q;

	xMsg68[12].Set		:=	OUT_CU.bMsg6812;(* B6812 reserve operating message 220 *) (*import HMI Extension *)
	MM2VIS.bMsg6812		:=	xMsg68[12].Q;

	xMsg68[13].Set		:=	OUT_CU.bMsg6813;(* B6813 reserve operating message 221 *) (*import HMI Extension *)
	MM2VIS.bMsg6813		:=	xMsg68[13].Q;

	xMsg68[14].Set		:=	OUT_CU.bMsg6814;(* B6814 reserve operating message 222 *) (*import HMI Extension *)
	MM2VIS.bMsg6814		:=	xMsg68[14].Q;

	xMsg68[15].Set		:=	OUT_CU.bMsg6815;(* B6815 reserve operating message 223 *) (*import HMI Extension *)
	MM2VIS.bMsg6815		:=	xMsg68[15].Q;

	xMsg68[16].Set		:=	OUT_CU.bMsg6816;(* B6816 reserve operating message 224 *) (*import HMI Extension *)
	MM2VIS.bMsg6816		:=	xMsg68[16].Q;

	xMsg68[17].Set		:=	OUT_CU.bMsg6817;(* B6817 reserve operating message 225 *) (*import HMI Extension *)
	MM2VIS.bMsg6817		:=	xMsg68[17].Q;

	xMsg68[18].Set		:=	OUT_CU.bMsg6818;(* B6818 reserve operating message 226 *) (*import HMI Extension *)
	MM2VIS.bMsg6818		:=	xMsg68[18].Q;

	xMsg68[19].Set		:=	OUT_CU.bMsg6819;(* B6819 reserve operating message 227 *) (*import HMI Extension *)
	MM2VIS.bMsg6819		:=	xMsg68[19].Q;

	xMsg68[20].Set		:=	OUT_CU.bMsg6820;(* B6820 reserve operating message 228 *) (*import HMI Extension *)
	MM2VIS.bMsg6820		:=	xMsg68[20].Q;

	xMsg68[21].Set		:=	OUT_CU.bMsg6821;(* B6821 reserve operating message 229 *) (*import HMI Extension *)
	MM2VIS.bMsg6821		:=	xMsg68[21].Q;

	xMsg68[22].Set		:=	OUT_CU.bMsg6822;(* B6822 reserve operating message 230 *) (*import HMI Extension *)
	MM2VIS.bMsg6822		:=	xMsg68[22].Q;

	xMsg68[23].Set		:=	OUT_CU.bMsg6823;(* B6823 reserve operating message 231 *) (*import HMI Extension *)
	MM2VIS.bMsg6823		:=	xMsg68[23].Q;

	xMsg68[24].Set		:=	OUT_CU.bMsg6824;(* B6824 reserve operating message 232 *) (*import HMI Extension *)
	MM2VIS.bMsg6824		:=	xMsg68[24].Q;

	xMsg68[25].Set		:=	OUT_CU.bMsg6825;(* B6825 reserve operating message 233 *) (*import HMI Extension *)
	MM2VIS.bMsg6825		:=	xMsg68[25].Q;

	xMsg68[26].Set		:=	OUT_CU.bMsg6826;(* B6826 reserve operating message 234 *) (*import HMI Extension *)
	MM2VIS.bMsg6826		:=	xMsg68[26].Q;

	xMsg68[27].Set		:=	OUT_CU.bMsg6827;(* B6827 reserve operating message 235 *) (*import HMI Extension *)
	MM2VIS.bMsg6827		:=	xMsg68[27].Q;

	xMsg68[28].Set		:=	OUT_CU.bMsg6828;(* B6828 reserve operating message 236 *) (*import HMI Extension *)
	MM2VIS.bMsg6828		:=	xMsg68[28].Q;

	xMsg68[29].Set		:=	OUT_CU.bMsg6829;(* B6829 reserve operating message 237 *) (*import HMI Extension *)
	MM2VIS.bMsg6829		:=	xMsg68[29].Q;

	xMsg68[30].Set		:=	OUT_CU.bMsg6830;(* B6830 reserve operating message 238 *) (*import HMI Extension *)
	MM2VIS.bMsg6830		:=	xMsg68[30].Q;

	xMsg68[31].Set		:=	OUT_CU.bMsg6831;(* B6831 reserve operating message 239 *) (*import HMI Extension *)
	MM2VIS.bMsg6831		:=	xMsg68[31].Q;

	xMsg68[32].Set		:=	OUT_CU.bMsg6832;(* B6832 reserve operating message 240 *) (*import HMI Extension *)
	MM2VIS.bMsg6832		:=	xMsg68[32].Q;

	xMsg68[33].Set		:=	OUT_CU.bMsg6833;(* B6833 reserve operating message 241 *) (*import HMI Extension *)
	MM2VIS.bMsg6833		:=	xMsg68[33].Q;

	xMsg68[34].Set		:=	OUT_CU.bMsg6834;(* B6834 reserve operating message 242 *) (*import HMI Extension *)
	MM2VIS.bMsg6834		:=	xMsg68[34].Q;

	xMsg68[35].Set		:=	OUT_CU.bMsg6835;(* B6835 reserve operating message 243 *) (*import HMI Extension *)
	MM2VIS.bMsg6835		:=	xMsg68[35].Q;

	xMsg68[36].Set		:=	OUT_CU.bMsg6836;(* B6836 reserve operating message 244 *) (*import HMI Extension *)
	MM2VIS.bMsg6836		:=	xMsg68[36].Q;

	xMsg68[37].Set		:=	OUT_CU.bMsg6837;(* B6837 reserve operating message 245 *) (*import HMI Extension *)
	MM2VIS.bMsg6837		:=	xMsg68[37].Q;

	xMsg68[38].Set		:=	OUT_CU.bMsg6838;(* B6838 reserve operating message 246 *) (*import HMI Extension *)
	MM2VIS.bMsg6838		:=	xMsg68[38].Q;

	xMsg68[39].Set		:=	OUT_CU.bMsg6839;(* B6839 reserve operating message 247 *) (*import HMI Extension *)
	MM2VIS.bMsg6839		:=	xMsg68[39].Q;

	xMsg68[40].Set		:=	OUT_CU.bMsg6840;(* B6840 reserve operating message 248 *) (*import HMI Extension *)
	MM2VIS.bMsg6840		:=	xMsg68[40].Q;

	xMsg68[41].Set		:=	OUT_CU.bMsg6841;(* B6841 reserve operating message 249 *) (*import HMI Extension *)
	MM2VIS.bMsg6841		:=	xMsg68[41].Q;

	xMsg68[42].Set		:=	OUT_CU.bMsg6842;(* B6842 reserve operating message 250 *) (*import HMI Extension *)
	MM2VIS.bMsg6842		:=	xMsg68[42].Q;

	xMsg68[43].Set		:=	OUT_CU.bMsg6843;(* B6843 reserve operating message 251 *) (*import HMI Extension *)
	MM2VIS.bMsg6843		:=	xMsg68[43].Q;

	xMsg68[44].Set		:=	OUT_CU.bMsg6844;(* B6844 reserve operating message 252 *) (*import HMI Extension *)
	MM2VIS.bMsg6844		:=	xMsg68[44].Q;

	xMsg68[45].Set		:=	OUT_CU.bMsg6845;(* B6845 reserve operating message 253 *) (*import HMI Extension *)
	MM2VIS.bMsg6845		:=	xMsg68[45].Q;

	xMsg68[46].Set		:=	OUT_CU.bMsg6846;(* B6846 reserve operating message 254 *) (*import HMI Extension *)
	MM2VIS.bMsg6846		:=	xMsg68[46].Q;

	xMsg68[47].Set		:=	OUT_CU.bMsg6847;(* B6847 reserve operating message 255 *) (*import HMI Extension *)
	MM2VIS.bMsg6847		:=	xMsg68[47].Q;

	xMsg68[48].Set		:=	OUT_CU.bMsg6848;(* B6848 reserve operating message 256 *) (*import HMI Extension *)
	MM2VIS.bMsg6848		:=	xMsg68[48].Q;

	xMsg68[49].Set		:=	OUT_CU.bMsg6849;(* B6849 reserve operating message 257 *) (*import HMI Extension *)
	MM2VIS.bMsg6849		:=	xMsg68[49].Q;

	xMsg68[50].Set		:=	OUT_CU.bMsg6850;(* B6850 reserve operating message 258 *) (*import HMI Extension *)
	MM2VIS.bMsg6850		:=	xMsg68[50].Q;

	xMsg68[51].Set		:=	OUT_CU.bMsg6851;(* B6851 reserve operating message 259 *) (*import HMI Extension *)
	MM2VIS.bMsg6851		:=	xMsg68[51].Q;

	xMsg68[52].Set		:=	OUT_CU.bMsg6852;(* B6852 reserve operating message 260 *) (*import HMI Extension *)
	MM2VIS.bMsg6852		:=	xMsg68[52].Q;

	xMsg68[53].Set		:=	OUT_CU.bMsg6853;(* B6853 reserve operating message 261 *) (*import HMI Extension *)
	MM2VIS.bMsg6853		:=	xMsg68[53].Q;

	xMsg68[54].Set		:=	OUT_CU.bMsg6854;(* B6854 reserve operating message 262 *) (*import HMI Extension *)
	MM2VIS.bMsg6854		:=	xMsg68[54].Q;

	xMsg68[55].Set		:=	OUT_CU.bMsg6855;(* B6855 reserve operating message 263 *) (*import HMI Extension *)
	MM2VIS.bMsg6855		:=	xMsg68[55].Q;

	xMsg68[56].Set		:=	OUT_CU.bMsg6856;(* B6856 reserve operating message 264 *) (*import HMI Extension *)
	MM2VIS.bMsg6856		:=	xMsg68[56].Q;

	xMsg68[57].Set		:=	OUT_CU.bMsg6857;(* B6857 reserve operating message 265 *) (*import HMI Extension *)
	MM2VIS.bMsg6857		:=	xMsg68[57].Q;

	xMsg68[58].Set		:=	OUT_CU.bMsg6858;(* B6858 reserve operating message 266 *) (*import HMI Extension *)
	MM2VIS.bMsg6858		:=	xMsg68[58].Q;

	xMsg68[59].Set		:=	OUT_CU.bMsg6859;(* B6859 reserve operating message 267 *) (*import HMI Extension *)
	MM2VIS.bMsg6859		:=	xMsg68[59].Q;

	xMsg68[60].Set		:=	OUT_CU.bMsg6860;(* B6860 reserve operating message 268 *) (*import HMI Extension *)
	MM2VIS.bMsg6860		:=	xMsg68[60].Q;

	xMsg68[61].Set		:=	OUT_CU.bMsg6861;(* B6861 reserve operating message 269 *) (*import HMI Extension *)
	MM2VIS.bMsg6861		:=	xMsg68[61].Q;

	xMsg68[62].Set		:=	OUT_CU.bMsg6862;(* B6862 reserve operating message 270 *) (*import HMI Extension *)
	MM2VIS.bMsg6862		:=	xMsg68[62].Q;

	xMsg68[63].Set		:=	OUT_CU.bMsg6863;(* B6863 reserve operating message 271 *) (*import HMI Extension *)
	MM2VIS.bMsg6863		:=	xMsg68[63].Q;

	xMsg68[64].Set		:=	OUT_CU.bMsg6864;(* B6864 reserve operating message 272 *) (*import HMI Extension *)
	MM2VIS.bMsg6864		:=	xMsg68[64].Q;

	xMsg68[65].Set		:=	OUT_CU.bMsg6865;(* B6865 reserve operating message 273 *) (*import HMI Extension *)
	MM2VIS.bMsg6865		:=	xMsg68[65].Q;

	xMsg68[66].Set		:=	OUT_CU.bMsg6866;(* B6866 reserve operating message 274 *) (*import HMI Extension *)
	MM2VIS.bMsg6866		:=	xMsg68[66].Q;

	xMsg68[67].Set		:=	OUT_CU.bMsg6867;(* B6867 reserve operating message 275 *) (*import HMI Extension *)
	MM2VIS.bMsg6867		:=	xMsg68[67].Q;

	xMsg68[68].Set		:=	OUT_CU.bMsg6868;(* B6868 reserve operating message 276 *) (*import HMI Extension *)
	MM2VIS.bMsg6868		:=	xMsg68[68].Q;

	xMsg68[69].Set		:=	OUT_CU.bMsg6869;(* B6869 reserve operating message 277 *) (*import HMI Extension *)
	MM2VIS.bMsg6869		:=	xMsg68[69].Q;

	xMsg68[70].Set		:=	OUT_CU.bMsg6870;(* B6870 reserve operating message 278 *) (*import HMI Extension *)
	MM2VIS.bMsg6870		:=	xMsg68[70].Q;

	xMsg68[71].Set		:=	OUT_CU.bMsg6871;(* B6871 reserve operating message 279 *) (*import HMI Extension *)
	MM2VIS.bMsg6871		:=	xMsg68[71].Q;

	xMsg68[72].Set		:=	OUT_CU.bMsg6872;(* B6872 reserve operating message 280 *) (*import HMI Extension *)
	MM2VIS.bMsg6872		:=	xMsg68[72].Q;

	xMsg68[73].Set		:=	OUT_CU.bMsg6873;(* B6873 reserve operating message 281 *) (*import HMI Extension *)
	MM2VIS.bMsg6873		:=	xMsg68[73].Q;

	xMsg68[74].Set		:=	OUT_CU.bMsg6874;(* B6874 reserve operating message 282 *) (*import HMI Extension *)
	MM2VIS.bMsg6874		:=	xMsg68[74].Q;

	xMsg68[75].Set		:=	OUT_CU.bMsg6875;(* B6875 reserve operating message 283 *) (*import HMI Extension *)
	MM2VIS.bMsg6875		:=	xMsg68[75].Q;

	xMsg68[76].Set		:=	OUT_CU.bMsg6876;(* B6876 reserve operating message 284 *) (*import HMI Extension *)
	MM2VIS.bMsg6876		:=	xMsg68[76].Q;

	xMsg68[77].Set		:=	OUT_CU.bMsg6877;(* B6877 reserve operating message 285 *) (*import HMI Extension *)
	MM2VIS.bMsg6877		:=	xMsg68[77].Q;

	xMsg68[78].Set		:=	OUT_CU.bMsg6878;(* B6878 reserve operating message 286 *) (*import HMI Extension *)
	MM2VIS.bMsg6878		:=	xMsg68[78].Q;

	xMsg68[79].Set		:=	OUT_CU.bMsg6879;(* B6879 reserve operating message 287 *) (*import HMI Extension *)
	MM2VIS.bMsg6879		:=	xMsg68[79].Q;

	xMsg68[80].Set		:=	OUT_CU.bMsg6880;(* B6880 reserve operating message 288 *) (*import HMI Extension *)
	MM2VIS.bMsg6880		:=	xMsg68[80].Q;

	xMsg68[81].Set		:=	OUT_CU.bMsg6881;(* B6881 reserve operating message 289 *) (*import HMI Extension *)
	MM2VIS.bMsg6881		:=	xMsg68[81].Q;

	xMsg68[82].Set		:=	OUT_CU.bMsg6882;(* B6882 reserve operating message 290 *) (*import HMI Extension *)
	MM2VIS.bMsg6882		:=	xMsg68[82].Q;

	xMsg68[83].Set		:=	OUT_CU.bMsg6883;(* B6883 reserve operating message 291 *) (*import HMI Extension *)
	MM2VIS.bMsg6883		:=	xMsg68[83].Q;

	xMsg68[84].Set		:=	OUT_CU.bMsg6884;(* B6884 reserve operating message 292 *) (*import HMI Extension *)
	MM2VIS.bMsg6884		:=	xMsg68[84].Q;

	xMsg68[85].Set		:=	OUT_CU.bMsg6885;(* B6885 reserve operating message 293 *) (*import HMI Extension *)
	MM2VIS.bMsg6885		:=	xMsg68[85].Q;

	xMsg68[86].Set		:=	OUT_CU.bMsg6886;(* B6886 reserve operating message 294 *) (*import HMI Extension *)
	MM2VIS.bMsg6886		:=	xMsg68[86].Q;

	xMsg68[87].Set		:=	OUT_CU.bMsg6887;(* B6887 reserve operating message 295 *) (*import HMI Extension *)
	MM2VIS.bMsg6887		:=	xMsg68[87].Q;

	xMsg68[88].Set		:=	OUT_CU.bMsg6888;(* B6888 reserve operating message 296 *) (*import HMI Extension *)
	MM2VIS.bMsg6888		:=	xMsg68[88].Q;

	xMsg68[89].Set		:=	OUT_CU.bMsg6889;(* B6889 reserve operating message 297 *) (*import HMI Extension *)
	MM2VIS.bMsg6889		:=	xMsg68[89].Q;

	xMsg68[90].Set		:=	OUT_CU.bMsg6890;(* B6890 reserve operating message 298 *) (*import HMI Extension *)
	MM2VIS.bMsg6890		:=	xMsg68[90].Q;

	xMsg68[91].Set		:=	OUT_CU.bMsg6891;(* B6891 reserve operating message 299 *) (*import HMI Extension *)
	MM2VIS.bMsg6891		:=	xMsg68[91].Q;

	xMsg68[92].Set		:=	OUT_CU.bMsg6892;(* B6892 reserve operating message 300 *) (*import HMI Extension *)
	MM2VIS.bMsg6892		:=	xMsg68[92].Q;

	xMsg68[93].Set		:=	OUT_CU.bMsg6893;(* B6893 reserve operating message 301 *) (*import HMI Extension *)
	MM2VIS.bMsg6893		:=	xMsg68[93].Q;

	xMsg68[94].Set		:=	OUT_CU.bMsg6894;(* B6894 reserve operating message 302 *) (*import HMI Extension *)
	MM2VIS.bMsg6894		:=	xMsg68[94].Q;

	xMsg68[95].Set		:=	OUT_CU.bMsg6895;(* B6895 reserve operating message 303 *) (*import HMI Extension *)
	MM2VIS.bMsg6895		:=	xMsg68[95].Q;

	xMsg68[96].Set		:=	OUT_CU.bMsg6896;(* B6896 reserve operating message 304 *) (*import HMI Extension *)
	MM2VIS.bMsg6896		:=	xMsg68[96].Q;

	xMsg68[97].Set		:=	OUT_CU.bMsg6897;(* B6897 reserve operating message 305 *) (*import HMI Extension *)
	MM2VIS.bMsg6897		:=	xMsg68[97].Q;

	xMsg68[98].Set		:=	OUT_CU.bMsg6898;(* B6898 reserve operating message 306 *) (*import HMI Extension *)
	MM2VIS.bMsg6898		:=	xMsg68[98].Q;

	xMsg68[99].Set		:=	OUT_CU.bMsg6899;(* B6899 reserve operating message 307 *) (*import HMI Extension *)
	MM2VIS.bMsg6899		:=	xMsg68[99].Q;

//OLD	xMsg68[100].Set		:=	OUT_CU.bMsgxxxx;(* B4200 reserve operating message 308 OLD, do not use*) (*import HMI Extension *)
//OLD	MM2VIS.bMsg4200		:=	xMsg41[100].Q;

	(*----------------------------------------------------------------------*)
	iDelay_MsgAutoReset_100ms 	:= LIMIT(0, TIME_TO_INT(Para.tiDelay_MsgAutoReset / 100), 32767);	(*To Do: missing prototype parameter *)
	IF Para.tiDelay_MsgAutoReset = 0 THEN Para.tiDelay_MsgAutoReset := T#01m; END_IF				(*To Do: missing prototype parameter *)
	(*----------------------------------------------------------------------*)

END_PROGRAM
```

#### MsgCUInit.st - Initialization code
```iecst
(*******************************************************************************
Msg_CU	 			 alarms generation MM_Customized

This code is confidential and proprietary to the INNIO Company.
It may not be used in any form, or reproduced in any manner,
without written permission of the INNIO Company.
Copyright, INNIO Company, 2019

Customized modifications: -
------------------------

History:
-------
V0.00.0	29.07.2011	lettenb.	new
V4.07.1	29.03.2019	Hohensinner	added Warnings: W9285, W9286, W9287
V4.11.1	20.01.2022	Zengerer	added Arrays: B67xx, B68xx, W87xx

Instructions for use:
--------------------
1) declare alarm with function block "Msg"

2) use template to create a new alarm, substitue 0000 by message number:

	xMsg0000.Num		:=	0000;					alarm number
	xMsg0000.AmmSysAdr	:=  iAdrAmmBase2MM;			do not change
	xMsg0000.AmmOutAdr	:=  iAdrMM2AmmBase;			do not change

3) 	set alarm number

Outstandings:
------------
(*******************************************************************************)
PROGRAM _INIT

	iAdrAmmBase2MM		:=  ADR(IN_CU.tAB2CU);
	iAdrMM2AmmBase		:=  ADR(OUT_CU.tCU2AB);

	(*---------------------------------------------------------------------------*)
	xMsg1001.Num		:=	1001;
	xMsg1001.AmmInAdr	:=  iAdrAmmBase2MM;
	xMsg1001.AmmOutAdr	:=  iAdrMM2AmmBase;

	xMsg1002.Num		:=	1002;
	xMsg1002.AmmInAdr	:=  iAdrAmmBase2MM;
	xMsg1002.AmmOutAdr	:=  iAdrMM2AmmBase;

	xMsg1003.Num		:=	1003;
	xMsg1003.AmmInAdr	:=  iAdrAmmBase2MM;
	xMsg1003.AmmOutAdr	:=  iAdrMM2AmmBase;

	xMsg1004.Num		:=	1004;
	xMsg1004.AmmInAdr	:=  iAdrAmmBase2MM;
	xMsg1004.AmmOutAdr	:=  iAdrMM2AmmBase;

	xMsg1005.Num		:=	1005;
	xMsg1005.AmmInAdr	:=  iAdrAmmBase2MM;
	xMsg1005.AmmOutAdr	:=  iAdrMM2AmmBase;

	xMsg1006.Num		:=	1006;
	xMsg1006.AmmInAdr	:=  iAdrAmmBase2MM;
	xMsg1006.AmmOutAdr	:=  iAdrMM2AmmBase;

	xMsg1007.Num		:=	1007;
	xMsg1007.AmmInAdr	:=  iAdrAmmBase2MM;
	xMsg1007.AmmOutAdr	:=  iAdrMM2AmmBase;

	xMsg1008.Num		:=	1008;
	xMsg1008.AmmInAdr	:=  iAdrAmmBase2MM;
	xMsg1008.AmmOutAdr	:=  iAdrMM2AmmBase;

	xMsg1009.Num		:=	1009;
	xMsg1009.AmmInAdr	:=  iAdrAmmBase2MM;
	xMsg1009.AmmOutAdr	:=  iAdrMM2AmmBase;

	xMsg1010.Num		:=	1010;
	xMsg1010.AmmInAdr	:=  iAdrAmmBase2MM;
	xMsg1010.AmmOutAdr	:=  iAdrMM2AmmBase;

	xMsg1011.Num		:=	1011;
	xMsg1011.AmmInAdr	:=  iAdrAmmBase2MM;
	xMsg1011.AmmOutAdr	:=  iAdrMM2AmmBase;

	xMsg1012.Num		:=	1012;
	xMsg1012.AmmInAdr	:=  iAdrAmmBase2MM;
	xMsg1012.AmmOutAdr	:=  iAdrMM2AmmBase;

	xMsg1013.Num		:=	1013;
	xMsg1013.AmmInAdr	:=  iAdrAmmBase2MM;
	xMsg1013.AmmOutAdr	:=  iAdrMM2AmmBase;

	xMsg1014.Num		:=	1014;
	xMsg1014.AmmInAdr	:=  iAdrAmmBase2MM;
	xMsg1014.AmmOutAdr	:=  iAdrMM2AmmBase;

	xMsg1015.Num		:=	1015;
	xMsg1015.AmmInAdr	:=  iAdrAmmBase2MM;
	xMsg1015.AmmOutAdr	:=  iAdrMM2AmmBase;

	xMsg1016.Num		:=	1016;
	xMsg1016.AmmInAdr	:=  iAdrAmmBase2MM;
	xMsg1016.AmmOutAdr	:=  iAdrMM2AmmBase;

	xMsg1177.Num		:=	1177;			(* W1177 Signal fail: reserve analog in 1 *)
	xMsg1177.AmmInAdr	:=  iAdrAmmBase2MM;
	xMsg1177.AmmOutAdr	:=  iAdrMM2AmmBase;

	xMsg1178.Num		:=	1178;			(* W1178 Signal fail: reserve analog in 2 *)
	xMsg1178.AmmInAdr	:=  iAdrAmmBase2MM;
	xMsg1178.AmmOutAdr	:=  iAdrMM2AmmBase;

	xMsg1179.Num		:=	1179;			(* W1179 Signal fail: reserve analog in 3 *)
	xMsg1179.AmmInAdr	:=  iAdrAmmBase2MM;
	xMsg1179.AmmOutAdr	:=  iAdrMM2AmmBase;

	xMsg1180.Num		:=	1180;			(* W1180 Signal fail: reserve analog in 4 *)
	xMsg1180.AmmInAdr	:=  iAdrAmmBase2MM;
	xMsg1180.AmmOutAdr	:=  iAdrMM2AmmBase;

	xMsg1181.Num		:=	1181;			(* W1181 Signal fail: reserve analog in 5 *)
	xMsg1181.AmmInAdr	:=  iAdrAmmBase2MM;
	xMsg1181.AmmOutAdr	:=  iAdrMM2AmmBase;

	xMsg1182.Num		:=	1182;			(* W1182 Signal fail: reserve analog in 6 *)
	xMsg1182.AmmInAdr	:=  iAdrAmmBase2MM;
	xMsg1182.AmmOutAdr	:=  iAdrMM2AmmBase;

	xMsg1183.Num		:=	1183;			(* W1183 Signal fail: reserve analog in 7 *)
	xMsg1183.AmmInAdr	:=  iAdrAmmBase2MM;
	xMsg1183.AmmOutAdr	:=  iAdrMM2AmmBase;

	xMsg1184.Num		:=	1184;			(* W1184 Signal fail: reserve analog in 8 *)
	xMsg1184.AmmInAdr	:=  iAdrAmmBase2MM;
	xMsg1184.AmmOutAdr	:=  iAdrMM2AmmBase;

	xMsg1193.Num		:=	1193;
	xMsg1193.AmmInAdr	:=  iAdrAmmBase2MM;
	xMsg1193.AmmOutAdr	:=  iAdrMM2AmmBase;

	xMsg1194.Num		:=	1194;
	xMsg1194.AmmInAdr	:=  iAdrAmmBase2MM;
	xMsg1194.AmmOutAdr	:=  iAdrMM2AmmBase;

	xMsg1195.Num		:=	1195;
	xMsg1195.AmmInAdr	:=  iAdrAmmBase2MM;
	xMsg1195.AmmOutAdr	:=  iAdrMM2AmmBase;

	xMsg1196.Num		:=	1196;
	xMsg1196.AmmInAdr	:=  iAdrAmmBase2MM;
	xMsg1196.AmmOutAdr	:=  iAdrMM2AmmBase;

	xMsg1197.Num		:=	1197;
	xMsg1197.AmmInAdr	:=  iAdrAmmBase2MM;
	xMsg1197.AmmOutAdr	:=  iAdrMM2AmmBase;

	xMsg1198.Num		:=	1198;
	xMsg1198.AmmInAdr	:=  iAdrAmmBase2MM;
	xMsg1198.AmmOutAdr	:=  iAdrMM2AmmBase;

	xMsg1199.Num		:=	1199;
	xMsg1199.AmmInAdr	:=  iAdrAmmBase2MM;
	xMsg1199.AmmOutAdr	:=  iAdrMM2AmmBase;

	xMsg1200.Num		:=	1200;
	xMsg1200.AmmInAdr	:=  iAdrAmmBase2MM;
	xMsg1200.AmmOutAdr	:=  iAdrMM2AmmBase;

	xMsg1201.Num		:=	1201;
	xMsg1201.AmmInAdr	:=  iAdrAmmBase2MM;
	xMsg1201.AmmOutAdr	:=  iAdrMM2AmmBase;

	xMsg1202.Num		:=	1202;
	xMsg1202.AmmInAdr	:=  iAdrAmmBase2MM;
	xMsg1202.AmmOutAdr	:=  iAdrMM2AmmBase;

	xMsg1203.Num		:=	1203;
	xMsg1203.AmmInAdr	:=  iAdrAmmBase2MM;
	xMsg1203.AmmOutAdr	:=  iAdrMM2AmmBase;

	xMsg1204.Num		:=	1204;
	xMsg1204.AmmInAdr	:=  iAdrAmmBase2MM;
	xMsg1204.AmmOutAdr	:=  iAdrMM2AmmBase;

	xMsg1205.Num		:=	1205;
	xMsg1205.AmmInAdr	:=  iAdrAmmBase2MM;
	xMsg1205.AmmOutAdr	:=  iAdrMM2AmmBase;

	xMsg1206.Num		:=	1206;
	xMsg1206.AmmInAdr	:=  iAdrAmmBase2MM;
	xMsg1206.AmmOutAdr	:=  iAdrMM2AmmBase;

	xMsg1207.Num		:=	1207;
	xMsg1207.AmmInAdr	:=  iAdrAmmBase2MM;
	xMsg1207.AmmOutAdr	:=  iAdrMM2AmmBase;

	xMsg1208.Num		:=	1208;
	xMsg1208.AmmInAdr	:=  iAdrAmmBase2MM;
	xMsg1208.AmmOutAdr	:=  iAdrMM2AmmBase;

	(*W1300, W1301 - W1399 Reserve AnalogIN 1-30*)
	(*moved*)
	(*W1400, W1401 - W1499 Reserve AnalogIN ...*)
	(*moved*)

	(*A1601, A1602 - A1700 additional Reserve ALARMS *)
	FOR cnt := 0 TO 100 DO								(*remark: index 0 element is not in use, but called here also, to avoid possible watch errors in some AS- versions *)
		xMsg16[cnt].Num			:=	1600+cnt;
		xMsg16[cnt].AmmInAdr	:=  iAdrAmmBase2MM;
		xMsg16[cnt].AmmOutAdr	:=  iAdrMM2AmmBase;
	END_FOR

	(*W1701, W1702 - W1800 additional Reserve WARNINGS *)
	FOR cnt := 0 TO 100 DO								(*remark: index 0 element is not in use, but called here also, to avoid possible watch errors in some AS- versions *)
		xMsg17[cnt].Num			:=	1700+cnt;
		xMsg17[cnt].AmmInAdr	:=  iAdrAmmBase2MM;
		xMsg17[cnt].AmmOutAdr	:=  iAdrMM2AmmBase;
	END_FOR

	xMsg2087.Num		:=	2087;
	xMsg2087.AmmInAdr	:=  iAdrAmmBase2MM;
	xMsg2087.AmmOutAdr	:=  iAdrMM2AmmBase;

	xMsg2088.Num		:=	2088;
	xMsg2088.AmmInAdr	:=  iAdrAmmBase2MM;
	xMsg2088.AmmOutAdr	:=  iAdrMM2AmmBase;

	xMsg2089.Num		:=	2089;
	xMsg2089.AmmInAdr	:=  iAdrAmmBase2MM;
	xMsg2089.AmmOutAdr	:=  iAdrMM2AmmBase;

	xMsg2090.Num		:=	2090;
	xMsg2090.AmmInAdr	:=  iAdrAmmBase2MM;
	xMsg2090.AmmOutAdr	:=  iAdrMM2AmmBase;

	xMsg2091.Num		:=	2091;
	xMsg2091.AmmInAdr	:=  iAdrAmmBase2MM;
	xMsg2091.AmmOutAdr	:=  iAdrMM2AmmBase;

	xMsg2092.Num		:=	2092;
	xMsg2092.AmmInAdr	:=  iAdrAmmBase2MM;
	xMsg2092.AmmOutAdr	:=  iAdrMM2AmmBase;

	xMsg2093.Num		:=	2093;
	xMsg2093.AmmInAdr	:=  iAdrAmmBase2MM;
	xMsg2093.AmmOutAdr	:=  iAdrMM2AmmBase;

	xMsg2094.Num		:=	2094;
	xMsg2094.AmmInAdr	:=  iAdrAmmBase2MM;
	xMsg2094.AmmOutAdr	:=  iAdrMM2AmmBase;

	xMsg2095.Num		:=	2095;
	xMsg2095.AmmInAdr	:=  iAdrAmmBase2MM;
	xMsg2095.AmmOutAdr	:=  iAdrMM2AmmBase;

	xMsg2096.Num		:=	2096;
	xMsg2096.AmmInAdr	:=  iAdrAmmBase2MM;
	xMsg2096.AmmOutAdr	:=  iAdrMM2AmmBase;

	(*- NETZBEZUGSREGLER --------------------------------------------------------------------*)

	xMsg2302.Num		:=	2302;
	xMsg2302.AmmInAdr	:=  iAdrAmmBase2MM;
	xMsg2302.AmmOutAdr	:=  iAdrMM2AmmBase;

	xMsg2303.Num		:=	2303;
	xMsg2303.AmmInAdr	:=  iAdrAmmBase2MM;
	xMsg2303.AmmOutAdr	:=  iAdrMM2AmmBase;

	xMsg2415.Num		:=	2415;
	xMsg2415.AmmInAdr	:=  iAdrAmmBase2MM;
	xMsg2415.AmmOutAdr	:=  iAdrMM2AmmBase;

	xMsg2416.Num		:=	2416;
	xMsg2416.AmmInAdr	:=  iAdrAmmBase2MM;
	xMsg2416.AmmOutAdr	:=  iAdrMM2AmmBase;

	xMsg2417.Num		:=	2417;
	xMsg2417.AmmInAdr	:=  iAdrAmmBase2MM;
	xMsg2417.AmmOutAdr	:=  iAdrMM2AmmBase;

	xMsg2418.Num		:=	2418;
	xMsg2418.AmmInAdr	:=  iAdrAmmBase2MM;
	xMsg2418.AmmOutAdr	:=  iAdrMM2AmmBase;

	xMsg2419.Num		:=	2419;
	xMsg2419.AmmInAdr	:=  iAdrAmmBase2MM;
	xMsg2419.AmmOutAdr	:=  iAdrMM2AmmBase;

	xMsg2420.Num		:=	2420;
	xMsg2420.AmmInAdr	:=  iAdrAmmBase2MM;
	xMsg2420.AmmOutAdr	:=  iAdrMM2AmmBase;

	(*************)

	xMsg3232.Num		:=	3232;
	xMsg3232.AmmInAdr	:=  iAdrAmmBase2MM;
	xMsg3232.AmmOutAdr	:=  iAdrMM2AmmBase;

	xMsg3233.Num		:=	3233;
	xMsg3233.AmmInAdr	:=  iAdrAmmBase2MM;
	xMsg3233.AmmOutAdr	:=  iAdrMM2AmmBase;

	xMsg3234.Num		:=	3234;
	xMsg3234.AmmInAdr	:=  iAdrAmmBase2MM;
	xMsg3234.AmmOutAdr	:=  iAdrMM2AmmBase;

	xMsg3235.Num		:=	3235;
	xMsg3235.AmmInAdr	:=  iAdrAmmBase2MM;
	xMsg3235.AmmOutAdr	:=  iAdrMM2AmmBase;

	xMsg3236.Num		:=	3236;
	xMsg3236.AmmInAdr	:=  iAdrAmmBase2MM;
	xMsg3236.AmmOutAdr	:=  iAdrMM2AmmBase;

	xMsg3237.Num		:=	3237;
	xMsg3237.AmmInAdr	:=  iAdrAmmBase2MM;
	xMsg3237.AmmOutAdr	:=  iAdrMM2AmmBase;

	xMsg3250.Num		:=	3250;
	xMsg3250.AmmInAdr	:=  iAdrAmmBase2MM;
	xMsg3250.AmmOutAdr	:=  iAdrMM2AmmBase;

	xMsg3251.Num		:=	3251;
	xMsg3251.AmmInAdr	:=  iAdrAmmBase2MM;
	xMsg3251.AmmOutAdr	:=  iAdrMM2AmmBase;

	(*************)

	xMsg3565.Num		:=	3565;
	xMsg3565.AmmInAdr	:=  iAdrAmmBase2MM;
	xMsg3565.AmmOutAdr	:=  iAdrMM2AmmBase;

	(*************)

	(*A8966 - A8999 Reserve AnalogIN Alarms *)
	(*moved*)

	(*************)

	(*B3601 - 3699 additional Reserve op.messages *)
	FOR cnt := 0 TO 100 DO								(*remark: index 0 element is not in use, but called here also, to avoid possible watch errors in some AS- versions *)
		xMsg36[cnt].Num			:=	3600+cnt;			(* bugfix 2018! *)
		xMsg36[cnt].AmmInAdr	:=  iAdrAmmBase2MM;
		xMsg36[cnt].AmmOutAdr	:=  iAdrMM2AmmBase;
	END_FOR

	xMsg3700.Num		:=	3700;
	xMsg3700.AmmInAdr	:=  iAdrAmmBase2MM;
	xMsg3700.AmmOutAdr	:=  iAdrMM2AmmBase;

	(*B6701 - 6800 additional Reserve op.messages *)	(*import HMI Extension *)
	FOR cnt := 0 TO 100 DO								(*remark: index 0 element is not in use, but called here also, to avoid possible watch errors in some AS- versions *)
		xMsg67[cnt].Num			:=	6700+cnt;
		xMsg67[cnt].AmmInAdr	:=  iAdrAmmBase2MM;
		xMsg67[cnt].AmmOutAdr	:=  iAdrMM2AmmBase;
	END_FOR

	(*B6800 - 6899 additional Reserve op.messages *)	(*import HMI Extension *)
	FOR cnt := 0 TO 99 DO								(*remark: index 100 element is not in use, but called here also, to avoid possible watch errors in some AS- versions *)
		xMsg68[cnt].Num			:=	6800+cnt;
		xMsg68[cnt].AmmInAdr	:=  iAdrAmmBase2MM;
		xMsg68[cnt].AmmOutAdr	:=  iAdrMM2AmmBase;
	END_FOR

	(*B8701 - 8799 additional Reserve WARNINGS *)		(*import HMI Extension *)
	FOR cnt := 0 TO 99 DO								(*remark: index 100 element is not in use, but called here also, to avoid possible watch errors in some AS- versions *)
		xMsg87[cnt].Num			:=	8700+cnt;
		xMsg87[cnt].AmmInAdr	:=  iAdrAmmBase2MM;
		xMsg87[cnt].AmmOutAdr	:=  iAdrMM2AmmBase;
	END_FOR

	(*************)

	xMsg9286.Num		:=	9286;
	xMsg9286.AmmInAdr	:=  iAdrAmmBase2MM;
	xMsg9286.AmmOutAdr	:=  iAdrMM2AmmBase;

	xMsg9287.Num		:=	9287;
	xMsg9287.AmmInAdr	:=  iAdrAmmBase2MM;
	xMsg9287.AmmOutAdr	:=  iAdrMM2AmmBase;

	(*************)

	(* OPERATING MESSAGES: *)
		OUT_CU.bMsg3232 :=		FALSE;	(* B3232 reserve operating message 1 *)
		OUT_CU.bMsg3233 :=		FALSE;	(* B3233 reserve operating message 2 *)
		OUT_CU.bMsg3234 :=		FALSE;	(* B3234 reserve operating message 3 *)
		OUT_CU.bMsg3235 :=		FALSE;	(* B3235 reserve operating message 4 *)
		OUT_CU.bMsg3236 := 		FALSE;	(* B3236 reserve operating message 5 *)
		OUT_CU.bMsg3237 := 		FALSE;	(* B3237 reserve operating message 6 *)

		OUT_CU.bMsg3250 := 		FALSE;	(* B3250 reserve operating message 7 *)
		OUT_CU.bMsg3251 := 		FALSE;	(* B3251 reserve operating message 8 *)

		OUT_CU.bMsg3601 := 		FALSE;	(* B3601 reserve operating message 9 *)
		OUT_CU.bMsg3602 := 		FALSE;	(* B3602 reserve operating message 10 *)
		OUT_CU.bMsg3603 := 		FALSE;	(* B3603 reserve operating message 11 *)
		OUT_CU.bMsg3604 := 		FALSE;	(* B3604 reserve operating message 12 *)
		OUT_CU.bMsg3605 := 		FALSE;	(* B3605 reserve operating message 13 *)
		OUT_CU.bMsg3606 := 		FALSE;	(* B3606 reserve operating message 14 *)
		OUT_CU.bMsg3607 := 		FALSE;	(* B3607 reserve operating message 15 *)
		OUT_CU.bMsg3608 := 		FALSE;	(* B3608 reserve operating message 16 *)
		OUT_CU.bMsg3609 := 		FALSE;	(* B3609 reserve operating message 17 *)
		OUT_CU.bMsg3610 := 		FALSE;	(* B3610 reserve operating message 18 *)

		OUT_CU.bMsg3611 := 		FALSE;	(* B3611 reserve operating message 19 *)
		OUT_CU.bMsg3612 := 		FALSE;	(*  	 reserve operating message 20 *)
		OUT_CU.bMsg3613 := 		FALSE;	(* 		 reserve operating message 21 *)
		OUT_CU.bMsg3614 := 		FALSE;	(* 		 reserve operating message 22 *)
		OUT_CU.bMsg3615 := 		FALSE;	(* 		 reserve operating message 23 *)
		OUT_CU.bMsg3616 := 		FALSE;	(* 		 reserve operating message 24 *)
		OUT_CU.bMsg3617 := 		FALSE;	(* 		 reserve operating message 25 *)
		OUT_CU.bMsg3618 := 		FALSE;	(* 		 reserve operating message 26 *)
		OUT_CU.bMsg3619 := 		FALSE;	(* 		 reserve operating message 27 *)
		OUT_CU.bMsg3620 := 		FALSE;	(* 		 reserve operating message 28 *)

		OUT_CU.bMsg3621 := 		FALSE;	(* B3621 reserve operating message 29 *)
		OUT_CU.bMsg3622 := 		FALSE;	(* 		 reserve operating message 30 *)
		OUT_CU.bMsg3623 := 		FALSE;	(* 		 reserve operating message 31 *)
		OUT_CU.bMsg3624 := 		FALSE;	(* 		 reserve operating message 32 *)
		OUT_CU.bMsg3625 := 		FALSE;	(* 		 reserve operating message 33 *)
		OUT_CU.bMsg3626 := 		FALSE;	(* 		 reserve operating message 34 *)
		OUT_CU.bMsg3627 := 		FALSE;	(* 		 reserve operating message 35 *)
		OUT_CU.bMsg3628 := 		FALSE;	(* 		 reserve operating message 36 *)
		OUT_CU.bMsg3629 := 		FALSE;	(* 		 reserve operating message 37 *)
		OUT_CU.bMsg3630 := 		FALSE;	(* 		 reserve operating message 38 *)

		OUT_CU.bMsg3631 := 		FALSE;	(* 		 reserve operating message 39 *)
		OUT_CU.bMsg3632 := 		FALSE;	(* 		 reserve operating message 40 *)
		OUT_CU.bMsg3633 := 		FALSE;	(* 		 reserve operating message 41 *)
		OUT_CU.bMsg3634 := 		FALSE;	(* 		 reserve operating message 42 *)
		OUT_CU.bMsg3635 := 		FALSE;	(* 		 reserve operating message 43 *)
		OUT_CU.bMsg3636 := 		FALSE;	(* 		 reserve operating message 44 *)
		OUT_CU.bMsg3637 := 		FALSE;	(* 		 reserve operating message 45 *)
		OUT_CU.bMsg3638 := 		FALSE;	(* 		 reserve operating message 46 *)
		OUT_CU.bMsg3639 := 		FALSE;	(* 		 reserve operating message 47 *)
		OUT_CU.bMsg3640 := 		FALSE;	(* 		 reserve operating message 48 *)

		OUT_CU.bMsg3641 := 		FALSE;	(* B3641 reserve operating message 49 *)
		OUT_CU.bMsg3642 := 		FALSE;	(* 		 reserve operating message 50 *)
		OUT_CU.bMsg3643 := 		FALSE;	(* 		 reserve operating message 51 *)
		OUT_CU.bMsg3644 := 		FALSE;	(* 		 reserve operating message 52 *)
		OUT_CU.bMsg3645 := 		FALSE;	(* 		 reserve operating message 53 *)
		OUT_CU.bMsg3646 := 		FALSE;	(* 		 reserve operating message 54 *)
		OUT_CU.bMsg3647 := 		FALSE;	(* 		 reserve operating message 55 *)
		OUT_CU.bMsg3648 := 		FALSE;	(* 		 reserve operating message 56 *)
		OUT_CU.bMsg3649 := 		FALSE;	(* 		 reserve operating message 57 *)
		OUT_CU.bMsg3650 := 		FALSE;	(* 		 reserve operating message 58 *)

		OUT_CU.bMsg3651 := 		FALSE;	(* 		 reserve operating message 59 *)
		OUT_CU.bMsg3652 := 		FALSE;	(* 		 reserve operating message 60 *)
		OUT_CU.bMsg3653 := 		FALSE;	(* 		 reserve operating message 61 *)
		OUT_CU.bMsg3654 := 		FALSE;	(* 		 reserve operating message 62 *)
		OUT_CU.bMsg3655 := 		FALSE;	(* 		 reserve operating message 63 *)
		OUT_CU.bMsg3656 := 		FALSE;	(* 		 reserve operating message 64 *)
		OUT_CU.bMsg3657 := 		FALSE;	(* 		 reserve operating message 65 *)
		OUT_CU.bMsg3658 := 		FALSE;	(* 		 reserve operating message 66 *)
		OUT_CU.bMsg3659 := 		FALSE;	(* 		 reserve operating message 67 *)
		OUT_CU.bMsg3660 := 		FALSE;	(* 		 reserve operating message 68 *)

		OUT_CU.bMsg3661 := 		FALSE;	(* B3661 reserve operating message 69 *)
		OUT_CU.bMsg3662 := 		FALSE;	(* 		 reserve operating message 70 *)
		OUT_CU.bMsg3663 := 		FALSE;	(* 		 reserve operating message 71 *)
		OUT_CU.bMsg3664 := 		FALSE;	(* 		 reserve operating message 72 *)
		OUT_CU.bMsg3665 := 		FALSE;	(* 		 reserve operating message 73 *)
		OUT_CU.bMsg3666 := 		FALSE;	(* 		 reserve operating message 74 *)
		OUT_CU.bMsg3667 := 		FALSE;	(* 		 reserve operating message 75 *)
		OUT_CU.bMsg3668 := 		FALSE;	(* 		 reserve operating message 76 *)
		OUT_CU.bMsg3669 := 		FALSE;	(* 		 reserve operating message 77 *)
		OUT_CU.bMsg3670 := 		FALSE;	(* 		 reserve operating message 78 *)

		OUT_CU.bMsg3671 := 		FALSE;	(* 		 reserve operating message 79 *)
		OUT_CU.bMsg3672 := 		FALSE;	(* 		 reserve operating message 80 *)
		OUT_CU.bMsg3673 := 		FALSE;	(* 		 reserve operating message 81 *)
		OUT_CU.bMsg3674 := 		FALSE;	(* 		 reserve operating message 82 *)
		OUT_CU.bMsg3675 := 		FALSE;	(* 		 reserve operating message 83 *)
		OUT_CU.bMsg3676 := 		FALSE;	(* 		 reserve operating message 84 *)
		OUT_CU.bMsg3677 := 		FALSE;	(* 		 reserve operating message 85 *)
		OUT_CU.bMsg3678 := 		FALSE;	(* 		 reserve operating message 86 *)
		OUT_CU.bMsg3679 := 		FALSE;	(* 		 reserve operating message 87 *)
		OUT_CU.bMsg3680 := 		FALSE;	(* 		 reserve operating message 88 *)

		OUT_CU.bMsg3681 := 		FALSE;	(* B3681 reserve operating message 89 *)
		OUT_CU.bMsg3682 := 		FALSE;	(* 		 reserve operating message 90 *)
		OUT_CU.bMsg3683 := 		FALSE;	(* 		 reserve operating message 91 *)
		OUT_CU.bMsg3684 := 		FALSE;	(* 		 reserve operating message 92 *)
		OUT_CU.bMsg3685 := 		FALSE;	(* 		 reserve operating message 93 *)
		OUT_CU.bMsg3686 := 		FALSE;	(* 		 reserve operating message 94 *)
		OUT_CU.bMsg3687 := 		FALSE;	(* 		 reserve operating message 95 *)
		OUT_CU.bMsg3688 := 		FALSE;	(* 		 reserve operating message 96 *)
		OUT_CU.bMsg3689 := 		FALSE;	(* 		 reserve operating message 97 *)
		OUT_CU.bMsg3690 := 		FALSE;	(* 		 reserve operating message 98 *)

		OUT_CU.bMsg3691 := 		FALSE;	(* 		 reserve operating message 99 *)
		OUT_CU.bMsg3692 := 		FALSE;	(* 		 reserve operating message 100 *)
		OUT_CU.bMsg3693 := 		FALSE;	(* 		 reserve operating message 101 *)
		OUT_CU.bMsg3694 := 		FALSE;	(* 		 reserve operating message 102 *)
		OUT_CU.bMsg3695 := 		FALSE;	(* 		 reserve operating message 103 *)
		OUT_CU.bMsg3696 := 		FALSE;	(* 		 reserve operating message 104 *)
		OUT_CU.bMsg3697 := 		FALSE;	(* 		 reserve operating message 105 *)
		OUT_CU.bMsg3698 := 		FALSE;	(* 		 reserve operating message 106 *)
		OUT_CU.bMsg3699 := 		FALSE;	(* 		 reserve operating message 107 *)
		OUT_CU.bMsg3700 := 		FALSE;	(* 		 reserve operating message 108 *)

		OUT_CU.bMsg6701 := 		FALSE;	(* B6701 reserve operating message 109 *) (*import HMI Extension *)
		OUT_CU.bMsg6702 := 		FALSE;	(* B6702 reserve operating message 110 *) (*import HMI Extension *)
		OUT_CU.bMsg6703 := 		FALSE;	(* B6703 reserve operating message 111 *) (*import HMI Extension *)
		OUT_CU.bMsg6704 := 		FALSE;	(* B6704 reserve operating message 112 *) (*import HMI Extension *)
		OUT_CU.bMsg6705 := 		FALSE;	(* B6705 reserve operating message 113 *) (*import HMI Extension *)
		OUT_CU.bMsg6706 := 		FALSE;	(* B6706 reserve operating message 114 *) (*import HMI Extension *)
		OUT_CU.bMsg6707 := 		FALSE;	(* B6707 reserve operating message 115 *) (*import HMI Extension *)
		OUT_CU.bMsg6708 := 		FALSE;	(* B6708 reserve operating message 116 *) (*import HMI Extension *)
		OUT_CU.bMsg6709 := 		FALSE;	(* B6709 reserve operating message 117 *) (*import HMI Extension *)
		OUT_CU.bMsg6710 := 		FALSE;	(* B6710 reserve operating message 118 *) (*import HMI Extension *)

		OUT_CU.bMsg6711 := 		FALSE;	(* B6711 reserve operating message 119 *) (*import HMI Extension *)
		OUT_CU.bMsg6712 := 		FALSE;	(* B6712 reserve operating message 120 *) (*import HMI Extension *)
		OUT_CU.bMsg6713 := 		FALSE;	(* B6713 reserve operating message 121 *) (*import HMI Extension *)
		OUT_CU.bMsg6714 := 		FALSE;	(* B6714 reserve operating message 122 *) (*import HMI Extension *)
		OUT_CU.bMsg6715 := 		FALSE;	(* B6715 reserve operating message 123 *) (*import HMI Extension *)
		OUT_CU.bMsg6716 := 		FALSE;	(* B6716 reserve operating message 124 *) (*import HMI Extension *)
		OUT_CU.bMsg6717 := 		FALSE;	(* B6717 reserve operating message 125 *) (*import HMI Extension *)
		OUT_CU.bMsg6718 := 		FALSE;	(* B6718 reserve operating message 126 *) (*import HMI Extension *)
		OUT_CU.bMsg6719 := 		FALSE;	(* B6719 reserve operating message 127 *) (*import HMI Extension *)
		OUT_CU.bMsg6720 := 		FALSE;	(* B6720 reserve operating message 128 *) (*import HMI Extension *)

		OUT_CU.bMsg6721 := 		FALSE;	(* B6721 reserve operating message 129 *) (*import HMI Extension *)
		OUT_CU.bMsg6722 := 		FALSE;	(* B6722 reserve operating message 130 *) (*import HMI Extension *)
		OUT_CU.bMsg6723 := 		FALSE;	(* B6723 reserve operating message 131 *) (*import HMI Extension *)
		OUT_CU.bMsg6724 := 		FALSE;	(* B6724 reserve operating message 132 *) (*import HMI Extension *)
		OUT_CU.bMsg6725 := 		FALSE;	(* B6725 reserve operating message 133 *) (*import HMI Extension *)
		OUT_CU.bMsg6726 := 		FALSE;	(* B6726 reserve operating message 134 *) (*import HMI Extension *)
		OUT_CU.bMsg6727 := 		FALSE;	(* B6727 reserve operating message 135 *) (*import HMI Extension *)
		OUT_CU.bMsg6728 := 		FALSE;	(* B6728 reserve operating message 136 *) (*import HMI Extension *)
		OUT_CU.bMsg6729 := 		FALSE;	(* B6729 reserve operating message 137 *) (*import HMI Extension *)
		OUT_CU.bMsg6730 := 		FALSE;	(* B6730 reserve operating message 138 *) (*import HMI Extension *)

		OUT_CU.bMsg6731 := 		FALSE;	(* B6731 reserve operating message 139 *) (*import HMI Extension *)
		OUT_CU.bMsg6732 := 		FALSE;	(* B6732 reserve operating message 140 *) (*import HMI Extension *)
		OUT_CU.bMsg6733 := 		FALSE;	(* B6733 reserve operating message 141 *) (*import HMI Extension *)
		OUT_CU.bMsg6734 := 		FALSE;	(* B6734 reserve operating message 142 *) (*import HMI Extension *)
		OUT_CU.bMsg6735 := 		FALSE;	(* B6735 reserve operating message 143 *) (*import HMI Extension *)
		OUT_CU.bMsg6736 := 		FALSE;	(* B6736 reserve operating message 144 *) (*import HMI Extension *)
		OUT_CU.bMsg6737 := 		FALSE;	(* B6737 reserve operating message 145 *) (*import HMI Extension *)
		OUT_CU.bMsg6738 := 		FALSE;	(* B6738 reserve operating message 146 *) (*import HMI Extension *)
		OUT_CU.bMsg6739 := 		FALSE;	(* B6739 reserve operating message 147 *) (*import HMI Extension *)
		OUT_CU.bMsg6740 := 		FALSE;	(* B6740 reserve operating message 148 *) (*import HMI Extension *)

		OUT_CU.bMsg6741 := 		FALSE;	(* B6741 reserve operating message 149 *) (*import HMI Extension *)
		OUT_CU.bMsg6742 := 		FALSE;	(* B6742 reserve operating message 150 *) (*import HMI Extension *)
		OUT_CU.bMsg6743 := 		FALSE;	(* B6743 reserve operating message 151 *) (*import HMI Extension *)
		OUT_CU.bMsg6744 := 		FALSE;	(* B6744 reserve operating message 152 *) (*import HMI Extension *)
		OUT_CU.bMsg6745 := 		FALSE;	(* B6745 reserve operating message 153 *) (*import HMI Extension *)
		OUT_CU.bMsg6746 := 		FALSE;	(* B6746 reserve operating message 154 *) (*import HMI Extension *)
		OUT_CU.bMsg6747 := 		FALSE;	(* B6747 reserve operating message 155 *) (*import HMI Extension *)
		OUT_CU.bMsg6748 := 		FALSE;	(* B6748 reserve operating message 156 *) (*import HMI Extension *)
		OUT_CU.bMsg6749 := 		FALSE;	(* B6749 reserve operating message 157 *) (*import HMI Extension *)
		OUT_CU.bMsg6750 := 		FALSE;	(* B6750 reserve operating message 158 *) (*import HMI Extension *)

		OUT_CU.bMsg6751 := 		FALSE;	(* B6751 reserve operating message 159 *) (*import HMI Extension *)
		OUT_CU.bMsg6752 := 		FALSE;	(* B6752 reserve operating message 160 *) (*import HMI Extension *)
		OUT_CU.bMsg6753 := 		FALSE;	(* B6753 reserve operating message 161 *) (*import HMI Extension *)
		OUT_CU.bMsg6754 := 		FALSE;	(* B6754 reserve operating message 162 *) (*import HMI Extension *)
		OUT_CU.bMsg6755 := 		FALSE;	(* B6755 reserve operating message 163 *) (*import HMI Extension *)
		OUT_CU.bMsg6756 := 		FALSE;	(* B6756 reserve operating message 164 *) (*import HMI Extension *)
		OUT_CU.bMsg6757 := 		FALSE;	(* B6757 reserve operating message 165 *) (*import HMI Extension *)
		OUT_CU.bMsg6758 := 		FALSE;	(* B6758 reserve operating message 166 *) (*import HMI Extension *)
		OUT_CU.bMsg6759 := 		FALSE;	(* B6759 reserve operating message 167 *) (*import HMI Extension *)
		OUT_CU.bMsg6760 := 		FALSE;	(* B6760 reserve operating message 168 *) (*import HMI Extension *)

		OUT_CU.bMsg6761 := 		FALSE;	(* B6761 reserve operating message 169 *) (*import HMI Extension *)
		OUT_CU.bMsg6762 := 		FALSE;	(* B6762 reserve operating message 170 *) (*import HMI Extension *)
		OUT_CU.bMsg6763 := 		FALSE;	(* B6763 reserve operating message 171 *) (*import HMI Extension *)
		OUT_CU.bMsg6764 := 		FALSE;	(* B6764 reserve operating message 172 *) (*import HMI Extension *)
		OUT_CU.bMsg6765 := 		FALSE;	(* B6765 reserve operating message 173 *) (*import HMI Extension *)
		OUT_CU.bMsg6766 := 		FALSE;	(* B6766 reserve operating message 174 *) (*import HMI Extension *)
		OUT_CU.bMsg6767 := 		FALSE;	(* B6767 reserve operating message 175 *) (*import HMI Extension *)
		OUT_CU.bMsg6768 := 		FALSE;	(* B6768 reserve operating message 176 *) (*import HMI Extension *)
		OUT_CU.bMsg6769 := 		FALSE;	(* B6769 reserve operating message 177 *) (*import HMI Extension *)
		OUT_CU.bMsg6770 := 		FALSE;	(* B6770 reserve operating message 178 *) (*import HMI Extension *)

		OUT_CU.bMsg6771 := 		FALSE;	(* B6771 reserve operating message 179 *) (*import HMI Extension *)
		OUT_CU.bMsg6772 := 		FALSE;	(* B6772 reserve operating message 180 *) (*import HMI Extension *)
		OUT_CU.bMsg6773 := 		FALSE;	(* B6773 reserve operating message 181 *) (*import HMI Extension *)
		OUT_CU.bMsg6774 := 		FALSE;	(* B6774 reserve operating message 182 *) (*import HMI Extension *)
		OUT_CU.bMsg6775 := 		FALSE;	(* B6775 reserve operating message 183 *) (*import HMI Extension *)
		OUT_CU.bMsg6776 := 		FALSE;	(* B6776 reserve operating message 184 *) (*import HMI Extension *)
		OUT_CU.bMsg6777 := 		FALSE;	(* B6777 reserve operating message 185 *) (*import HMI Extension *)
		OUT_CU.bMsg6778 := 		FALSE;	(* B6778 reserve operating message 186 *) (*import HMI Extension *)
		OUT_CU.bMsg6779 := 		FALSE;	(* B6779 reserve operating message 187 *) (*import HMI Extension *)
		OUT_CU.bMsg6780 := 		FALSE;	(* B6780 reserve operating message 188 *) (*import HMI Extension *)

		OUT_CU.bMsg6781 := 		FALSE;	(* B6781 reserve operating message 189 *) (*import HMI Extension *)
		OUT_CU.bMsg6782 := 		FALSE;	(* B6782 reserve operating message 190 *) (*import HMI Extension *)
		OUT_CU.bMsg6783 := 		FALSE;	(* B6783 reserve operating message 191 *) (*import HMI Extension *)
		OUT_CU.bMsg6784 := 		FALSE;	(* B6784 reserve operating message 192 *) (*import HMI Extension *)
		OUT_CU.bMsg6785 := 		FALSE;	(* B6785 reserve operating message 193 *) (*import HMI Extension *)
		OUT_CU.bMsg6786 := 		FALSE;	(* B6786 reserve operating message 194 *) (*import HMI Extension *)
		OUT_CU.bMsg6787 := 		FALSE;	(* B6787 reserve operating message 195 *) (*import HMI Extension *)
		OUT_CU.bMsg6788 := 		FALSE;	(* B6788 reserve operating message 196 *) (*import HMI Extension *)
		OUT_CU.bMsg6789 := 		FALSE;	(* B6789 reserve operating message 197 *) (*import HMI Extension *)
		OUT_CU.bMsg6790 := 		FALSE;	(* B6790 reserve operating message 198 *) (*import HMI Extension *)

		OUT_CU.bMsg6791 := 		FALSE;	(* B6791 reserve operating message 199 *) (*import HMI Extension *)
		OUT_CU.bMsg6792 := 		FALSE;	(* B6792 reserve operating message 200 *) (*import HMI Extension *)
		OUT_CU.bMsg6793 := 		FALSE;	(* B6793 reserve operating message 201 *) (*import HMI Extension *)
		OUT_CU.bMsg6794 := 		FALSE;	(* B6794 reserve operating message 202 *) (*import HMI Extension *)
		OUT_CU.bMsg6795 := 		FALSE;	(* B6795 reserve operating message 203 *) (*import HMI Extension *)
		OUT_CU.bMsg6796 := 		FALSE;	(* B6796 reserve operating message 204 *) (*import HMI Extension *)
		OUT_CU.bMsg6797 := 		FALSE;	(* B6797 reserve operating message 205 *) (*import HMI Extension *)
		OUT_CU.bMsg6798 := 		FALSE;	(* B6798 reserve operating message 206 *) (*import HMI Extension *)
		OUT_CU.bMsg6799 := 		FALSE;	(* B6799 reserve operating message 207 *) (*import HMI Extension *)
		OUT_CU.bMsg6800 := 		FALSE;	(* B6800 reserve operating message 208 *) (*import HMI Extension *)

		OUT_CU.bMsg6801 := 		FALSE;	(* B6801 reserve operating message 209 *) (*import HMI Extension *)
		OUT_CU.bMsg6802 := 		FALSE;	(* B6802 reserve operating message 210 *) (*import HMI Extension *)
		OUT_CU.bMsg6803 := 		FALSE;	(* B6803 reserve operating message 211 *) (*import HMI Extension *)
		OUT_CU.bMsg6804 := 		FALSE;	(* B6804 reserve operating message 212 *) (*import HMI Extension *)
		OUT_CU.bMsg6805 := 		FALSE;	(* B6805 reserve operating message 213 *) (*import HMI Extension *)
		OUT_CU.bMsg6806 := 		FALSE;	(* B6806 reserve operating message 214 *) (*import HMI Extension *)
		OUT_CU.bMsg6807 := 		FALSE;	(* B6807 reserve operating message 215 *) (*import HMI Extension *)
		OUT_CU.bMsg6808 := 		FALSE;	(* B6808 reserve operating message 216 *) (*import HMI Extension *)
		OUT_CU.bMsg6809 := 		FALSE;	(* B6809 reserve operating message 217 *) (*import HMI Extension *)
		OUT_CU.bMsg6810 := 		FALSE;	(* B6810 reserve operating message 218 *) (*import HMI Extension *)

		OUT_CU.bMsg6811 := 		FALSE;	(* B6811 reserve operating message 219 *) (*import HMI Extension *)
		OUT_CU.bMsg6812 := 		FALSE;	(* B6812 reserve operating message 220 *) (*import HMI Extension *)
		OUT_CU.bMsg6813 := 		FALSE;	(* B6813 reserve operating message 221 *) (*import HMI Extension *)
		OUT_CU.bMsg6814 := 		FALSE;	(* B6814 reserve operating message 222 *) (*import HMI Extension *)
		OUT_CU.bMsg6815 := 		FALSE;	(* B6815 reserve operating message 223 *) (*import HMI Extension *)
		OUT_CU.bMsg6816 := 		FALSE;	(* B6816 reserve operating message 224 *) (*import HMI Extension *)
		OUT_CU.bMsg6817 := 		FALSE;	(* B6817 reserve operating message 225 *) (*import HMI Extension *)
		OUT_CU.bMsg6818 := 		FALSE;	(* B6818 reserve operating message 226 *) (*import HMI Extension *)
		OUT_CU.bMsg6819 := 		FALSE;	(* B6819 reserve operating message 227 *) (*import HMI Extension *)
		OUT_CU.bMsg6820 := 		FALSE;	(* B6820 reserve operating message 228 *) (*import HMI Extension *)

		OUT_CU.bMsg6821 := 		FALSE;	(* B6821 reserve operating message 229 *) (*import HMI Extension *)
		OUT_CU.bMsg6822 := 		FALSE;	(* B6822 reserve operating message 230 *) (*import HMI Extension *)
		OUT_CU.bMsg6823 := 		FALSE;	(* B6823 reserve operating message 231 *) (*import HMI Extension *)
		OUT_CU.bMsg6824 := 		FALSE;	(* B6824 reserve operating message 232 *) (*import HMI Extension *)
		OUT_CU.bMsg6825 := 		FALSE;	(* B6825 reserve operating message 233 *) (*import HMI Extension *)
		OUT_CU.bMsg6826 := 		FALSE;	(* B6826 reserve operating message 234 *) (*import HMI Extension *)
		OUT_CU.bMsg6827 := 		FALSE;	(* B6827 reserve operating message 235 *) (*import HMI Extension *)
		OUT_CU.bMsg6828 := 		FALSE;	(* B6828 reserve operating message 236 *) (*import HMI Extension *)
		OUT_CU.bMsg6829 := 		FALSE;	(* B6829 reserve operating message 237 *) (*import HMI Extension *)
		OUT_CU.bMsg6830 := 		FALSE;	(* B6830 reserve operating message 238 *) (*import HMI Extension *)

		OUT_CU.bMsg6831 := 		FALSE;	(* B6831 reserve operating message 239 *) (*import HMI Extension *)
		OUT_CU.bMsg6832 := 		FALSE;	(* B6832 reserve operating message 240 *) (*import HMI Extension *)
		OUT_CU.bMsg6833 := 		FALSE;	(* B6833 reserve operating message 241 *) (*import HMI Extension *)
		OUT_CU.bMsg6834 := 		FALSE;	(* B6834 reserve operating message 242 *) (*import HMI Extension *)
		OUT_CU.bMsg6835 := 		FALSE;	(* B6835 reserve operating message 243 *) (*import HMI Extension *)
		OUT_CU.bMsg6836 := 		FALSE;	(* B6836 reserve operating message 244 *) (*import HMI Extension *)
		OUT_CU.bMsg6837 := 		FALSE;	(* B6837 reserve operating message 245 *) (*import HMI Extension *)
		OUT_CU.bMsg6838 := 		FALSE;	(* B6838 reserve operating message 246 *) (*import HMI Extension *)
		OUT_CU.bMsg6839 := 		FALSE;	(* B6839 reserve operating message 247 *) (*import HMI Extension *)
		OUT_CU.bMsg6840 := 		FALSE;	(* B6840 reserve operating message 248 *) (*import HMI Extension *)

		OUT_CU.bMsg6841 := 		FALSE;	(* B6841 reserve operating message 249 *) (*import HMI Extension *)
		OUT_CU.bMsg6842 := 		FALSE;	(* B6842 reserve operating message 250 *) (*import HMI Extension *)
		OUT_CU.bMsg6843 := 		FALSE;	(* B6843 reserve operating message 251 *) (*import HMI Extension *)
		OUT_CU.bMsg6844 := 		FALSE;	(* B6844 reserve operating message 252 *) (*import HMI Extension *)
		OUT_CU.bMsg6845 := 		FALSE;	(* B6845 reserve operating message 253 *) (*import HMI Extension *)
		OUT_CU.bMsg6846 := 		FALSE;	(* B6846 reserve operating message 254 *) (*import HMI Extension *)
		OUT_CU.bMsg6847 := 		FALSE;	(* B6847 reserve operating message 255 *) (*import HMI Extension *)
		OUT_CU.bMsg6848 := 		FALSE;	(* B6848 reserve operating message 256 *) (*import HMI Extension *)
		OUT_CU.bMsg6849 := 		FALSE;	(* B6849 reserve operating message 257 *) (*import HMI Extension *)
		OUT_CU.bMsg6850 := 		FALSE;	(* B6850 reserve operating message 258 *) (*import HMI Extension *)

		OUT_CU.bMsg6851 := 		FALSE;	(* B6851 reserve operating message 259 *) (*import HMI Extension *)
		OUT_CU.bMsg6852 := 		FALSE;	(* B6852 reserve operating message 260 *) (*import HMI Extension *)
		OUT_CU.bMsg6853 := 		FALSE;	(* B6853 reserve operating message 261 *) (*import HMI Extension *)
		OUT_CU.bMsg6854 := 		FALSE;	(* B6854 reserve operating message 262 *) (*import HMI Extension *)
		OUT_CU.bMsg6855 := 		FALSE;	(* B6855 reserve operating message 263 *) (*import HMI Extension *)
		OUT_CU.bMsg6856 := 		FALSE;	(* B6856 reserve operating message 264 *) (*import HMI Extension *)
		OUT_CU.bMsg6857 := 		FALSE;	(* B6857 reserve operating message 265 *) (*import HMI Extension *)
		OUT_CU.bMsg6858 := 		FALSE;	(* B6858 reserve operating message 266 *) (*import HMI Extension *)
		OUT_CU.bMsg6859 := 		FALSE;	(* B6859 reserve operating message 267 *) (*import HMI Extension *)
		OUT_CU.bMsg6860 := 		FALSE;	(* B6860 reserve operating message 268 *) (*import HMI Extension *)

		OUT_CU.bMsg6861 := 		FALSE;	(* B6861 reserve operating message 269 *) (*import HMI Extension *)
		OUT_CU.bMsg6862 := 		FALSE;	(* B6862 reserve operating message 270 *) (*import HMI Extension *)
		OUT_CU.bMsg6863 := 		FALSE;	(* B6863 reserve operating message 271 *) (*import HMI Extension *)
		OUT_CU.bMsg6864 := 		FALSE;	(* B6864 reserve operating message 272 *) (*import HMI Extension *)
		OUT_CU.bMsg6865 := 		FALSE;	(* B6865 reserve operating message 273 *) (*import HMI Extension *)
		OUT_CU.bMsg6866 := 		FALSE;	(* B6866 reserve operating message 274 *) (*import HMI Extension *)
		OUT_CU.bMsg6867 := 		FALSE;	(* B6867 reserve operating message 275 *) (*import HMI Extension *)
		OUT_CU.bMsg6868 := 		FALSE;	(* B6868 reserve operating message 276 *) (*import HMI Extension *)
		OUT_CU.bMsg6869 := 		FALSE;	(* B6869 reserve operating message 277 *) (*import HMI Extension *)
		OUT_CU.bMsg6870 := 		FALSE;	(* B6870 reserve operating message 278 *) (*import HMI Extension *)

		OUT_CU.bMsg6871 := 		FALSE;	(* B6871 reserve operating message 279 *) (*import HMI Extension *)
		OUT_CU.bMsg6872 := 		FALSE;	(* B6872 reserve operating message 280 *) (*import HMI Extension *)
		OUT_CU.bMsg6873 := 		FALSE;	(* B6873 reserve operating message 281 *) (*import HMI Extension *)
		OUT_CU.bMsg6874 := 		FALSE;	(* B6874 reserve operating message 282 *) (*import HMI Extension *)
		OUT_CU.bMsg6875 := 		FALSE;	(* B6875 reserve operating message 283 *) (*import HMI Extension *)
		OUT_CU.bMsg6876 := 		FALSE;	(* B6876 reserve operating message 284 *) (*import HMI Extension *)
		OUT_CU.bMsg6877 := 		FALSE;	(* B6877 reserve operating message 285 *) (*import HMI Extension *)
		OUT_CU.bMsg6878 := 		FALSE;	(* B6878 reserve operating message 286 *) (*import HMI Extension *)
		OUT_CU.bMsg6879 := 		FALSE;	(* B6879 reserve operating message 287 *) (*import HMI Extension *)
		OUT_CU.bMsg6880 := 		FALSE;	(* B6880 reserve operating message 288 *) (*import HMI Extension *)

		OUT_CU.bMsg6881 := 		FALSE;	(* B6881 reserve operating message 289 *) (*import HMI Extension *)
		OUT_CU.bMsg6882 := 		FALSE;	(* B6882 reserve operating message 290 *) (*import HMI Extension *)
		OUT_CU.bMsg6883 := 		FALSE;	(* B6883 reserve operating message 291 *) (*import HMI Extension *)
		OUT_CU.bMsg6884 := 		FALSE;	(* B6884 reserve operating message 292 *) (*import HMI Extension *)
		OUT_CU.bMsg6885 := 		FALSE;	(* B6885 reserve operating message 293 *) (*import HMI Extension *)
		OUT_CU.bMsg6886 := 		FALSE;	(* B6886 reserve operating message 294 *) (*import HMI Extension *)
		OUT_CU.bMsg6887 := 		FALSE;	(* B6887 reserve operating message 295 *) (*import HMI Extension *)
		OUT_CU.bMsg6888 := 		FALSE;	(* B6888 reserve operating message 296 *) (*import HMI Extension *)
		OUT_CU.bMsg6889 := 		FALSE;	(* B6889 reserve operating message 297 *) (*import HMI Extension *)
		OUT_CU.bMsg6890 := 		FALSE;	(* B6890 reserve operating message 298 *) (*import HMI Extension *)

		OUT_CU.bMsg6891 := 		FALSE;	(* B6891 reserve operating message 299 *) (*import HMI Extension *)
		OUT_CU.bMsg6892 := 		FALSE;	(* B6892 reserve operating message 300 *) (*import HMI Extension *)
		OUT_CU.bMsg6893 := 		FALSE;	(* B6893 reserve operating message 301 *) (*import HMI Extension *)
		OUT_CU.bMsg6894 := 		FALSE;	(* B6894 reserve operating message 302 *) (*import HMI Extension *)
		OUT_CU.bMsg6895 := 		FALSE;	(* B6895 reserve operating message 303 *) (*import HMI Extension *)
		OUT_CU.bMsg6896 := 		FALSE;	(* B6896 reserve operating message 304 *) (*import HMI Extension *)
		OUT_CU.bMsg6897 := 		FALSE;	(* B6897 reserve operating message 305 *) (*import HMI Extension *)
		OUT_CU.bMsg6898 := 		FALSE;	(* B6898 reserve operating message 306 *) (*import HMI Extension *)
		OUT_CU.bMsg6899 := 		FALSE;	(* B6899 reserve operating message 307 *) (*import HMI Extension *)
//OLD do not use		OUT_CU.bMsg4200 := 		FALSE;	(* B4200 reserve operating message 308 *) (*import HMI Extension *)

END_PROGRAM
```

#### MsgCU.var - Local variables
```iecst
(********************************************************************
 * COPYRIGHT -- INNIO Company
 ********************************************************************
 * Program: MsgCU
 * File: MsgCU.var
 * Author: 320003156
 * Created: November 24, 2011
 ********************************************************************
 * Local variables of program MsgCU
 ********************************************************************)
VAR
	xMsg2302 : Msg;
	xMsg2303 : Msg;
	xMsg2415 : Msg;
	xMsg2416 : Msg;
	xMsg2417 : Msg;
	xMsg2418 : Msg;
	xMsg2419 : Msg;
	xMsg2420 : Msg;
	xMsg1001 : Msg;
	xMsg1002 : Msg;
	xMsg1003 : Msg;
	xMsg1004 : Msg;
	xMsg1005 : Msg;
	xMsg1006 : Msg;
	xMsg1007 : Msg;
	xMsg1008 : Msg;
	xMsg1009 : Msg;
	xMsg1010 : Msg;
	xMsg1011 : Msg;
	xMsg1012 : Msg;
	xMsg1013 : Msg;
	xMsg1014 : Msg;
	xMsg1015 : Msg;
	xMsg1016 : Msg;
	xMsg1177 : Msg;
	xMsg1178 : Msg;
	xMsg1179 : Msg;
	xMsg1180 : Msg;
	xMsg1181 : Msg;
	xMsg1182 : Msg;
	xMsg1183 : Msg;
	xMsg1184 : Msg;
	xMsg1193 : Msg;
	xMsg1194 : Msg;
	xMsg1195 : Msg;
	xMsg1196 : Msg;
	xMsg1197 : Msg;
	xMsg1198 : Msg;
	xMsg1199 : Msg;
	xMsg1200 : Msg;
	xMsg1201 : Msg;
	xMsg1202 : Msg;
	xMsg1203 : Msg;
	xMsg1204 : Msg;
	xMsg1205 : Msg;
	xMsg1206 : Msg;
	xMsg1207 : Msg;
	xMsg1208 : Msg;
	xMsg2087 : Msg;
	xMsg2088 : Msg;
	xMsg2089 : Msg;
	xMsg2090 : Msg;
	xMsg2091 : Msg;
	xMsg2092 : Msg;
	xMsg2093 : Msg;
	xMsg2094 : Msg;
	xMsg2095 : Msg;
	xMsg2096 : Msg;
	xMsg3232 : Msg;
	xMsg3233 : Msg;
	xMsg3234 : Msg;
	xMsg3235 : Msg;
	xMsg3236 : Msg;
	xMsg3237 : Msg;
	xMsg3250 : Msg;
	xMsg3251 : Msg;
	xMsg3565 : Msg;
	xMsg36 : ARRAY[0..100] OF Msg;
	xMsg3700 : Msg;
	xMsg9286 : Msg;
	xMsg9287 : Msg;
	iAdrAmmBase2MM : UDINT;
	iAdrMM2AmmBase : UDINT;
	xMsg16 : ARRAY[0..100] OF Msg; (*Array of Msg for Reserve WARNINGS (element 0 not in use)*)
	xMsg17 : ARRAY[0..100] OF Msg; (*Array of Msg for Reserve WARNINGS (element 0 not in use)*)
	xMsg67 : ARRAY[0..100] OF Msg; (*Array of Msg for Reserve OPERATING Message (element 0 not in use) * import HMI Extension*)
	xMsg68 : ARRAY[0..100] OF Msg; (*Array of Msg for Reserve OPERATING Message (element 100 not in use) * import HMI Extension*)
	xMsg87 : ARRAY[0..100] OF Msg; (*Array of Msg for Reserve WARNINGS (element 100 not in use) * import HMI Extension*)
	TP_EngDSS_Mains_Off : TP;
	TP_EngDSS_Mains : TP;
	bCtr_Mns_Options_1 : BOOL; (*Debug only*)
	bCtr_Mns_Options_2 : BOOL; (*Debug only*)
	bCtr_Mns_Options_3 : BOOL; (*Debug only*)
	bCtr_Mns_Options_4 : BOOL; (*Debug only*)
	bCtr_Mns_Options_5 : BOOL; (*Debug only*)
	bCtr_Mns_Options_6 : BOOL; (*Debug only*)
	bCtr_Mns_Options_7 : BOOL; (*Debug only*)
	bCtr_Mns_Options_8 : BOOL; (*Debug only*)
	bCtr_Mns_Options_9 : BOOL; (*Debug only*)
	bCtr_Mns_Options_0 : BOOL; (*Debug only*)
	R_TRIG_Options : R_TRIG := (0);
	iDelay_MsgAutoReset_100ms : INT; (*Default Op Message Hold Time until Auto Reset*)
	iReset_Msg2419 : INT; (*internal timer counter*)
	iReset_Msg2420 : INT; (*internal timer counter*)
	iReset_Msg3232 : INT; (*internal timer counter*)
	iReset_Msg3233 : INT; (*internal timer counter*)
	iReset_Msg3234 : INT; (*internal timer counter*)
	iReset_Msg3235 : INT; (*internal timer counter*)
	iReset_Msg3236 : INT; (*internal timer counter*)
	iReset_Msg3237 : INT; (*internal timer counter*)
	iReset_Msg3250 : INT; (*internal timer counter*)
	iReset_Msg3251 : INT; (*internal timer counter*)
	iReset_Msg3700 : INT; (*internal timer counter*)
	iReset_Msg36 : ARRAY[0..99] OF INT; (*internal timer counter*)
	iReset_Msg67 : ARRAY[0..100] OF INT; (*internal timer counter * import HMI Extension*)
	iReset_Msg68 : ARRAY[0..100] OF INT; (*internal timer counter * import HMI Extension*)
	iReset_Msg2302 : INT; (*internal timer counter*)
	iReset_Msg2303 : INT; (*internal timer counter*)
END_VAR
```

### Program Logical/Customized/VisCU (IEC, version 4.04.0) - interface task for visualization adoptions

#### VisCUCyclic.st
```iecst
(*******************************************************************************
vis			visualization

This code is confidential AND proprietary to the INNIO Company.
It may NOT be used in any form, or reproduced in any manner,
without the express written permission of the INNIO Company.
Copyright, INNIO Company, 2019

Customized modifications: -
------------------------

History:
-------
V3.90.0	04.06.2013	Zengerer	new
V4.03.0	09.11.2015	Zengerer	Add Init file
V4.04.0	20.06.2016  Weitzer		add at MM2VIS & VIS2MM types rCustVis[33..50], bCustVis[33..50]

Instructions FOR use:
--------------------
Placeholders as reminder for VIS-tags from other tasks;
Add aditional function here as needed customized

Outstandings:
------------
*******************************************************************************)
PROGRAM _CYCLIC

	(* VIS2MM *)
	(*Counter inputs for user edit*)
	VIS2MM.iCount1;
	VIS2MM.iCount20;
	VIS2MM.iMaintenanceCount1;
	VIS2MM.iMaintenanceCount8;

	(*---------------------------------------------------------------------------*)
	(* MM2VIS *)
	(* Counters: *)
	MM2VIS.iCount1;
	MM2VIS.iCount2;
	MM2VIS.iCount3;
	MM2VIS.iCount4;
	MM2VIS.iCount5;
	MM2VIS.iCount6;
	MM2VIS.iCount7;
	MM2VIS.iCount8;
	MM2VIS.iCount9;
	MM2VIS.iCount10;
	MM2VIS.iCount11;
	MM2VIS.iCount12;
	MM2VIS.iCount13;
	MM2VIS.iCount14;
	MM2VIS.iCount15;
	MM2VIS.iCount16;
	MM2VIS.iCount17;
	MM2VIS.iCount18;
	MM2VIS.iCount19;
	MM2VIS.iCount20;

	MM2VIS.iMaintenanceCount1;
	MM2VIS.iMaintenanceCount2;
	MM2VIS.iMaintenanceCount3;
	MM2VIS.iMaintenanceCount4;
	MM2VIS.iMaintenanceCount5;
	MM2VIS.iMaintenanceCount6;
	MM2VIS.iMaintenanceCount7;
	MM2VIS.iMaintenanceCount8;

	(*Reserve alarms and warnings*)
	MM2VIS.bCustAlarm_Tripped[1];
	MM2VIS.bCustAlarm_Tripped[16];
	MM2VIS.bCustWarn_Tripped[1];
	MM2VIS.bCustWarn_Tripped[16];

	(*Reserve analog input channels*)
	MM2VIS.rCustAnaIn[1];
	MM2VIS.rCustAnaIn[2];
	MM2VIS.rCustAnaIn[3];
	MM2VIS.rCustAnaIn[4];
	MM2VIS.rCustAnaIn[5];
	MM2VIS.rCustAnaIn[6];
	MM2VIS.rCustAnaIn[7];
	MM2VIS.rCustAnaIn[8];
	MM2VIS.rCustAnaIn[9];
	MM2VIS.rCustAnaIn[10];
	MM2VIS.rCustAnaIn[11];
	MM2VIS.rCustAnaIn[12];
	MM2VIS.rCustAnaIn[13];
	MM2VIS.rCustAnaIn[14];
	MM2VIS.rCustAnaIn[15];
	MM2VIS.rCustAnaIn[16];
	MM2VIS.rCustAnaIn[32];

	(*CustomerIO channels*)
	MM2VIS.bUniDig[1];
	MM2VIS.rUniAna[1];

	(*-----------------------------------------------------------------------------*)
	(* 50 spare analog variables from PLC --> VISU *)
	MM2VIS.rCustVis[1];
	MM2VIS.rCustVis[2];
	MM2VIS.rCustVis[3];
	(*.....*)

	(* 50 spare digital variables from PLC --> VISU *)
	MM2VIS.bCustVis[1];
	MM2VIS.bCustVis[2];
	MM2VIS.bCustVis[3];
	(*.....*)

	(* 50 spare analog variables from VISU --> PLC *)
	VIS2MM.rCustVis[1];
	VIS2MM.rCustVis[2];
	VIS2MM.rCustVis[3];
	(*.....*)

	(* 50 spare digital variables from VISU --> PLC *)
	VIS2MM.bCustVis[1];
	VIS2MM.bCustVis[2];
	VIS2MM.bCustVis[3];
	(*.....*)

	(* Display process step info and remaining step time information at VIS   (Prototype) *)
	xOpMode(in:= IN_CU.iSt_OpMode);				(*get local representation of operating state*)

	IN_CU.iProcessStepTime;		(* 	Step Time Display	new with V4.04, 2016	*)
 	IN_CU.iIdx_ProcessStep;		(*	Step Time Display	new with V4.04, 2016 	*)

	OUT_CU.iIdx_ProcessStep_CU := IN_CU.iIdx_ProcessStep_AG; 	(*	 	Optional step information to display on VIS from module AG	 	*)
	OUT_CU.iProcessStepTime_CU := IN_CU.iProcessStepTime_AG; 	(*	 	Optional step time  info to display on VIS from module AG	 	 *)

	IF IN_CU.iIdx_ProcessStep > 0 THEN
		OUT_CU.iIdx_ProcessStep_CU := IN_CU.iIdx_ProcessStep;
		OUT_CU.iProcessStepTime_CU := IN_CU.iProcessStepTime;
	END_IF	// ELSE 	OUT_CU.iIdx_ProcessStep := IN_CU.iSt_OpMode;  END_IF

	(*-> See also MM Opstate: Para.iProcessStepInfo_Type[35];				=Parameter Array to control Step Info Visibility and Style 0=invisible; 1= allways visible; (+future options possible, e.g. user level?) *)

	//Task part was MOVED TO MM Opstate:
//	IF IN_CU.iProcessStepTime > 0 THEN
//		MM2VIS.iProcessStepTime := IN_CU.iProcessStepTime;
//	ELSE
//		IF MM2VIS.iIdx_ProcessStep = iIdx_ProcessStep_Last AND			(* detect state change*)
//		   NOT IN_CU.tImp_OpHour.Do	THEN					   			(* detect new operating hour *)
//			MM2VIS.iProcessStepTime := MM2VIS.iProcessStepTime + BOOL_TO_DINT(bSecondTic);	(* count seconds in same state *)
//		ELSE
//			MM2VIS.iProcessStepTime := 0;
//			iIdx_ProcessStep_Last := MM2VIS.iIdx_ProcessStep;
//		END_IF
//	END_IF
//
//	IF tRealTime.second = iRealTime_LastSecond THEN						(*to generate second tic*)
//		bSecondTic := FALSE;
//	ELSE
//		bSecondTic := TRUE;
//		iRealTime_LastSecond := tRealTime.second;
//	END_IF
//
//
//
//	MM2VIS.iIdx_ProcessStep;		(*ToDo: add custoized modifications here *)
//	MM2VIS.iProcessStepTime;		(*ToDo: add custoized modifications here *)
//
//	iProcessStepInfo_Last;

END_PROGRAM
```

#### VisCUInit.st
```iecst
(*******************************************************************************
vis	INIT		visualization

This code is confidential and proprietary to the INNIO Company.
It may not be used in any form, or reproduced in any manner,
without the express written permission of the INNIO Company.
Copyright, INNIO Company, 2019
*******************************************************************************)

PROGRAM _INIT

	(*-----------------------------------------------------------------------------*)
	bNoInitDetected := FALSE; 	 (* Insert this line into every tasks INIT code to activate download detection *)
END_PROGRAM
```

### Package Logical/Customized/Cust_Internals - tasks with no need for editing

### Program Logical/Customized/Cust_Internals/PermCU (IEC, version 4.06.0) - + storage of spare counter values ...

- PermCUCyclic.st (not readable text: treated as protected, skipped)

- PermCUInit.st (not readable text: treated as protected, skipped)

#### PermCU.var
```iecst
VAR
	tParaIntern : ParaHandler_typ; (*Connector type to perm_par*)
	bWriteDataObj : BOOL; (* TRUE=write data object module *)
	bDataObjLenErr : BOOL; (*Error occured in permem: data module size missmatch*)
	bCreateDataObj : BOOL; (* TRUE=create new data object *)
	bTest : BOOL; (*for development only*)
	write_once : BOOL; (* write permanent memory once *)
	DatObjCreate_01 : DatObjCreate; (* data object create *)
	DatObjInfo_01 : DatObjInfo; (* data object info *)
	DatObjRead_01 : DatObjRead; (* data object read *)
	DatObjWrite_01 : DatObjWrite; (* data object write *)
	ModuleName : STRING[35]; (* module name of object *)
	TON_WritePMEM : TON; (* delay write permanent memory *)
	ulPMPointer : UDINT; (* adress of actual checksum value *)
	ulChecksum : UDINT; (* parameter checksum value *)
	pm_len : UDINT; (* permanent value lenght *)
	ulChecksumOld : UDINT; (* last vlaue of parameter checksum *)
	ulChkValue : UDINT; (* actual value of parameter pointer *)
	pm_id : UDINT; (* permanent value identifier *)
	pm_p : UDINT; (* permanent value pointer *)
END_VAR
VAR CONSTANT
	ERR_NOERROR : UINT := 0;
END_VAR
VAR
	pm_Error : UINT; (* permanent value error *) (* Deleted: pm : ParaMem_typ; permanent memory tags mathias, 22.8.11*)
	ulAdrName : UDINT; (*Adress of string variable with metamodule name*)
	TON_BlockMinFileAge : TON; (*waiting time without file write after successful performed write*)
	bBlock_MinFileAge : BOOL := FALSE; (*pause the perm file write after each sucessful write*)
	iPM_WriteCnt : UDINT; (* *) (*old VarName: usPMWriteCnt*)
	iPM_WriteCnt_IncreaseValue : DINT := 1; (*Testkonstante +1*)
END_VAR
```

### Program Logical/Customized/Cust_Internals/BaseVers (IEC, version 4.08.0) - + readout info from file aeprot

- BaseVers.st (not readable text: treated as protected, skipped)

#### BaseVers.var
```iecst
VAR
	DatObjInfo_META : DatObjInfo;
	DatObjRead_META : DatObjRead;
	szMetaDataRaw : STRING[1000];
	szMetaData : ARRAY[0..3] OF STRING[35];
	ssIndex : INT;
	ssCount : INT;
	ucMetaDataRaw : ARRAY[0..1000] OF USINT;
	ssCount2 : INT;
	szMetaDataFile : STRING[35];
	pm_Error : UDINT; (* permanent value error *) (* Deleted: pm : ParaMem_typ; permanent memory tags mathias, 22.8.11*)
	bReadOutMETA_Once : BOOL;
END_VAR
VAR CONSTANT
	ERR_NOERROR : UINT := 0;
END_VAR
```

### Program Logical/Customized/Cust_Internals/ParCU (IEC, version 4.06.0) - + parameter storage and handling

- perm_par.st (not readable text: treated as protected, skipped)
